T_Surge_detection:=maskbitFunction(Trip_BITs_64_to_79,0);
T_VGD_fault :=maskbitFunction(Trip_BITs_64_to_79,1);
T_Long_time_PRV :=maskbitFunction(Trip_BITs_64_to_79,2);
T_Comp_thrust_bearing_position :=maskbitFunction(Trip_BITs_64_to_79,3);
T_Comp_thrust_neg_move:=maskbitFunction(Trip_BITs_64_to_79,4);
T_Comp_thrust_pos_move:=maskbitFunction(Trip_BITs_64_to_79,5);
S_Spare_1:=maskbitFunction(Trip_BITs_64_to_79,6);
S_Spare_1:=maskbitFunction(Trip_BITs_64_to_79,7);
S_Spare_1:=maskbitFunction(Trip_BITs_64_to_79,8);
S_Spare_1:=maskbitFunction(Trip_BITs_64_to_79,9);
S_Spare_1:=maskbitFunction(Trip_BITs_64_to_79,10);
S_Spare_1:=maskbitFunction(Trip_BITs_64_to_79,11);
S_Spare_1:=maskbitFunction(Trip_BITs_64_to_79,12);
S_Spare_1:=maskbitFunction(Trip_BITs_64_to_79,13);
S_Spare_1:=maskbitFunction(Trip_BITs_64_to_79,14);
S_Spare_1:=maskbitFunction(Trip_BITs_64_to_79,15);

T_Sensor_low_signal_AI_64 :=maskbitFunction(Trip_BITs_80_to_95,0);
T_Sensor_high_signal_AI_64 :=maskbitFunction(Trip_BITs_80_to_95,1);
T_Sensor_low_signal_AI_66 :=maskbitFunction(Trip_BITs_80_to_95,2);
T_Sensor_high_signal_AI_66 :=maskbitFunction(Trip_BITs_80_to_95,3);
//T_Sensor_low_signal_AI_116:=maskbitFunction(Trip_BITs_80_to_95,4);
//T_Sensor_high_signal_AI_116:=maskbitFunction(Trip_BITs_80_to_95,5);
//T_Sensor_low_signal_AI_118:=maskbitFunction(Trip_BITs_80_to_95,6);
//T_Sensor_high_signal_AI_118:=maskbitFunction(Trip_BITs_80_to_95,7);
T_Sensor_low_signal_AI_128 :=maskbitFunction(Trip_BITs_80_to_95,8);
T_Sensor_high_signal_AI_128 :=maskbitFunction(Trip_BITs_80_to_95,9);
T_Sensor_low_signal_AI_130 :=maskbitFunction(Trip_BITs_80_to_95,10);
T_Sensor_high_signal_AI_130 :=maskbitFunction(Trip_BITs_80_to_95,11);
T_Sensor_low_signal_AI_132 :=maskbitFunction(Trip_BITs_80_to_95,12);
T_Sensor_high_signal_AI_132 :=maskbitFunction(Trip_BITs_80_to_95,13);
T_Sensor_low_signal_AI_134 :=maskbitFunction(Trip_BITs_80_to_95,14);
T_Sensor_high_signal_AI_134 :=maskbitFunction(Trip_BITs_80_to_95,15);

T_Sensor_low_signal_AI_136 :=maskbitFunction(Trip_BITs_96_to_121,0);
T_Sensor_high_signal_AI_136 :=maskbitFunction(Trip_BITs_96_to_121,1);
T_Sensor_low_signal_AI_138 :=maskbitFunction(Trip_BITs_96_to_121,2);
T_Sensor_high_signal_AI_138 :=maskbitFunction(Trip_BITs_96_to_121,3);
T_Sensor_low_signal_AI_140 :=maskbitFunction(Trip_BITs_96_to_121,4);
T_Sensor_high_signal_AI_140 :=maskbitFunction(Trip_BITs_96_to_121,5);
T_Sensor_low_signal_AI_142 :=maskbitFunction(Trip_BITs_96_to_121,6);
T_Sensor_high_signal_AI_142 :=maskbitFunction(Trip_BITs_96_to_121,7);
T_Sensor_low_signal_AI_144 :=maskbitFunction(Trip_BITs_96_to_121,8);
T_Sensor_high_signal_AI_144 :=maskbitFunction(Trip_BITs_96_to_121,9);
T_Sensor_low_signal_AI_146 :=maskbitFunction(Trip_BITs_96_to_121,10);
T_Sensor_high_signal_AI_146 :=maskbitFunction(Trip_BITs_96_to_121,11);
T_Sensor_low_signal_AI_148 :=maskbitFunction(Trip_BITs_96_to_121,12);
T_Sensor_high_signal_AI_148 :=maskbitFunction(Trip_BITs_96_to_121,13);
T_Sensor_low_signal_AI_150 :=maskbitFunction(Trip_BITs_96_to_121,14);
T_Sensor_high_signal_AI_150 :=maskbitFunction(Trip_BITs_96_to_121,15);

T_Sensor_low_signal_AI_152 :=maskbitFunction(Trip_BITs_122_to_137,0);
T_Sensor_high_signal_AI_152 :=maskbitFunction(Trip_BITs_122_to_137,1);
T_Sensor_low_signal_AI_154 :=maskbitFunction(Trip_BITs_122_to_137,2);
T_Sensor_high_signal_AI_154 :=maskbitFunction(Trip_BITs_122_to_137,3);
T_Sensor_low_signal_AI_156 :=maskbitFunction(Trip_BITs_122_to_137,4);
T_Sensor_high_signal_AI_156 :=maskbitFunction(Trip_BITs_122_to_137,5);
T_Sensor_low_signal_AI_158 :=maskbitFunction(Trip_BITs_122_to_137,6);
T_Sensor_high_signal_AI_158 :=maskbitFunction(Trip_BITs_122_to_137,7);
T_Sensor_low_signal_AI_160 :=maskbitFunction(Trip_BITs_122_to_137,8);
T_Sensor_high_signal_AI_160 :=maskbitFunction(Trip_BITs_122_to_137,9);
T_Sensor_low_signal_AI_162 :=maskbitFunction(Trip_BITs_122_to_137,10);
T_Sensor_high_signal_AI_162 :=maskbitFunction(Trip_BITs_122_to_137,11);
T_Sensor_low_signal_AI_164 :=maskbitFunction(Trip_BITs_122_to_137,12);
T_Sensor_high_signal_AI_164 :=maskbitFunction(Trip_BITs_122_to_137,13);
T_Sensor_low_signal_AI_166 :=maskbitFunction(Trip_BITs_122_to_137,14);
T_Sensor_high_signal_AI_166 :=maskbitFunction(Trip_BITs_122_to_137,15);

T_Sensor_low_signal_AI_168 :=maskbitFunction(Trip_BITs_138_to_153,0);
T_Sensor_high_signal_AI_168 :=maskbitFunction(Trip_BITs_138_to_153,1);
T_Sensor_low_signal_AI_170 :=maskbitFunction(Trip_BITs_138_to_153,2);
T_Sensor_high_signal_AI_170:=maskbitFunction(Trip_BITs_138_to_153,3);
T_Sensor_low_signal_AI_172:=maskbitFunction(Trip_BITs_138_to_153,4);
T_Sensor_high_signal_AI_172:=maskbitFunction(Trip_BITs_138_to_153,5);
T_Sensor_low_signal_AI_174:=maskbitFunction(Trip_BITs_138_to_153,6);
T_Sensor_high_signal_AI_174:=maskbitFunction(Trip_BITs_138_to_153,7);
T_Sensor_low_signal_AI_176:=maskbitFunction(Trip_BITs_138_to_153,8);
T_Sensor_high_signal_AI_176:=maskbitFunction(Trip_BITs_138_to_153,9);
T_Sensor_low_signal_AI_178:=maskbitFunction(Trip_BITs_138_to_153,10);
T_Sensor_high_signal_AI_178:=maskbitFunction(Trip_BITs_138_to_153,11);
T_Sensor_low_signal_AI_180:=maskbitFunction(Trip_BITs_138_to_153,12);
T_Sensor_high_signal_AI_180:=maskbitFunction(Trip_BITs_138_to_153,13);
T_Sensor_low_signal_AI_182:=maskbitFunction(Trip_BITs_138_to_153,14);
T_Sensor_high_signal_AI_182:=maskbitFunction(Trip_BITs_138_to_153,15);

T_Sensor_low_signal_AI_184 :=maskbitFunction(Trip_BITs_154_to_169,0);
T_Sensor_high_signal_AI_184 :=maskbitFunction(Trip_BITs_154_to_169,1);
T_Sensor_low_signal_AI_186 :=maskbitFunction(Trip_BITs_154_to_169,2);
T_Sensor_high_signal_AI_186 :=maskbitFunction(Trip_BITs_154_to_169,3);
T_Sensor_low_signal_AI_188 :=maskbitFunction(Trip_BITs_154_to_169,4);
T_Sensor_high_signal_AI_188 :=maskbitFunction(Trip_BITs_154_to_169,5);
T_Sensor_low_signal_AI_190 :=maskbitFunction(Trip_BITs_154_to_169,6);
T_Sensor_high_signal_AI_190 :=maskbitFunction(Trip_BITs_154_to_169,7);
T_Sensor_low_signal_AI_192 :=maskbitFunction(Trip_BITs_154_to_169,8);
T_Sensor_high_signal_AI_192 :=maskbitFunction(Trip_BITs_154_to_169,9);
T_Sensor_low_signal_AI_194 :=maskbitFunction(Trip_BITs_154_to_169,10);
T_Sensor_high_signal_AI_194 :=maskbitFunction(Trip_BITs_154_to_169,11);
T_Sensor_low_signal_AI_196 :=maskbitFunction(Trip_BITs_154_to_169,12);
T_Sensor_high_signal_AI_196 :=maskbitFunction(Trip_BITs_154_to_169,13);
T_Sensor_low_signal_AI_198 :=maskbitFunction(Trip_BITs_154_to_169,14);
T_Sensor_high_signal_AI_198 :=maskbitFunction(Trip_BITs_154_to_169,15);

T_Sensor_low_signal_AI_200 :=maskbitFunction(Trip_BITs_170_to_185,0);
T_Sensor_high_signal_AI_200 :=maskbitFunction(Trip_BITs_170_to_185,1);
T_Sensor_low_signal_AI_202 :=maskbitFunction(Trip_BITs_170_to_185,2);
T_Sensor_high_signal_AI_202 :=maskbitFunction(Trip_BITs_170_to_185,3);
T_Sensor_low_signal_AI_204 :=maskbitFunction(Trip_BITs_170_to_185,4);
T_Sensor_high_signal_AI_204 :=maskbitFunction(Trip_BITs_170_to_185,5);
T_Sensor_low_signal_AI_206 :=maskbitFunction(Trip_BITs_170_to_185,6);
T_Sensor_high_signal_AI_206 :=maskbitFunction(Trip_BITs_170_to_185,7);
S_Spare_1:=maskbitFunction(Trip_BITs_170_to_185,8);
S_Spare_1 :=maskbitFunction(Trip_BITs_170_to_185,9);
S_Spare_1 :=maskbitFunction(Trip_BITs_170_to_185,10);
S_Spare_1 :=maskbitFunction(Trip_BITs_170_to_185,11);
S_Spare_1 :=maskbitFunction(Trip_BITs_170_to_185,12);
S_Spare_1 :=maskbitFunction(Trip_BITs_170_to_185,13);
S_Spare_1 :=maskbitFunction(Trip_BITs_170_to_185,14);
S_Spare_1 :=maskbitFunction(Trip_BITs_170_to_185,15);

T_Transformer_winding_temp :=maskbitFunction(Trip_BITs_186_to_201,0);
T_trafo_opening_main_breaker :=maskbitFunction(Trip_BITs_186_to_201,1);
S_Spare_1 :=maskbitFunction(Trip_BITs_186_to_201,2);
S_Spare_1 :=maskbitFunction(Trip_BITs_186_to_201,3);
S_Spare_1 :=maskbitFunction(Trip_BITs_186_to_201,4);
S_Spare_1 :=maskbitFunction(Trip_BITs_186_to_201,5);
S_Spare_1 :=maskbitFunction(Trip_BITs_186_to_201,6);
S_Spare_1 :=maskbitFunction(Trip_BITs_186_to_201,7);
S_Spare_1 :=maskbitFunction(Trip_BITs_186_to_201,8);
S_Spare_1 :=maskbitFunction(Trip_BITs_186_to_201,9);
S_Spare_1 :=maskbitFunction(Trip_BITs_186_to_201,10);
S_Spare_1 :=maskbitFunction(Trip_BITs_186_to_201,11);
S_Spare_1 :=maskbitFunction(Trip_BITs_186_to_201,12);
S_Spare_1 :=maskbitFunction(Trip_BITs_186_to_201,13);
S_Spare_1 :=maskbitFunction(Trip_BITs_186_to_201,14);
S_Spare_1 :=maskbitFunction(Trip_BITs_186_to_201,15);


// Alarm bits
A_low_disch_press:=maskbitFunction(Alarm_BITs_0_to_15,0);
A_high_disch_press:=maskbitFunction(Alarm_BITs_0_to_15,1);
A_Low_suction_pressure:=maskbitFunction(Alarm_BITs_0_to_15,2);
A_High_suction_pressure:=maskbitFunction(Alarm_BITs_0_to_15,3);
A_Low_press_ratio:=maskbitFunction(Alarm_BITs_0_to_15,4);
A_High_discharge_temp :=maskbitFunction(Alarm_BITs_0_to_15,5);
A_Low_discharge_superheat:=maskbitFunction(Alarm_BITs_0_to_15,6);
A_High_discharge_superheat:=maskbitFunction(Alarm_BITs_0_to_15,7);
S_Spare_1:=maskbitFunction(Alarm_BITs_0_to_15,8);
S_Spare_1:=maskbitFunction(Alarm_BITs_0_to_15,9);
A_Low_temp_oil_inlet_comp:=maskbitFunction(Alarm_BITs_0_to_15,10);
A_High_temp_oil_inlet_comp:=maskbitFunction(Alarm_BITs_0_to_15,11);
A_Low_oil_temp_receiver:=maskbitFunction(Alarm_BITs_0_to_15,12);
A_High_oil_temp_receiver:=maskbitFunction(Alarm_BITs_0_to_15,13);
A_Low_oil_diff_pressure:=maskbitFunction(Alarm_BITs_0_to_15,14);
A_High_oil_diff_pressure:=maskbitFunction(Alarm_BITs_0_to_15,15);

A_High_oil_filter_diff_press:=maskbitFunction(Alarm_BITs_16_to_31,0);
S_Spare_1:=maskbitFunction(Alarm_BITs_16_to_31,1);
S_Spare_1:=maskbitFunction(Alarm_BITs_16_to_31,2);
A_Low_CW_outlet_temp:=maskbitFunction(Alarm_BITs_16_to_31,3);
A_High_CW_inlet_temp:=maskbitFunction(Alarm_BITs_16_to_31,4);
A_Low_CW_dP:=maskbitFunction(Alarm_BITs_16_to_31,5);
A_High_CW_dP:=maskbitFunction(Alarm_BITs_16_to_31,6);
S_Spare_1:=maskbitFunction(Alarm_BITs_16_to_31,7);
S_Spare_1:=maskbitFunction(Alarm_BITs_16_to_31,8);
A_Low_SW_inlet_temp:=maskbitFunction(Alarm_BITs_16_to_31,9);
A_High_SW_inlet_temp:=maskbitFunction(Alarm_BITs_16_to_31,10);
A_Low_SW_dP:=maskbitFunction(Alarm_BITs_16_to_31,11);
A_High_SW_dP:=maskbitFunction(Alarm_BITs_16_to_31,12);
A_Low_liquid_level:=maskbitFunction(Alarm_BITs_16_to_31,13);
A_Seawater_pump_not_running:=maskbitFunction(Alarm_BITs_16_to_31,14);
S_Spare_1:=maskbitFunction(Alarm_BITs_16_to_31,15);

S_Spare_1:=maskbitFunction(Alarm_BITs_32_to_47,0);
A_High_motor_wind_temp_R:=maskbitFunction(Alarm_BITs_32_to_47,1);
A_High_motor_wind_temp_S:=maskbitFunction(Alarm_BITs_32_to_47,2);
A_High_motor_wind_temp_T:=maskbitFunction(Alarm_BITs_32_to_47,3);
A_High_comp_mo_DE_bear_temp:=maskbitFunction(Alarm_BITs_32_to_47,4);
A_High_comp_mo_NDE_bear_temp:=maskbitFunction(Alarm_BITs_32_to_47,5);
A_High_motor_air_temp:=maskbitFunction(Alarm_BITs_32_to_47,6); 
A_High_comp_mo_DE_bear_vib:=maskbitFunction(Alarm_BITs_32_to_47,7);
A_High_comp_mo_NDE_bear_vib:=maskbitFunction(Alarm_BITs_32_to_47,8);
S_Spare_1:=maskbitFunction(Alarm_BITs_32_to_47,9);
S_Spare_1:=maskbitFunction(Alarm_BITs_32_to_47,10);
A_VGD_fault:=maskbitFunction(Alarm_BITs_32_to_47,11);
A_High_control_panel_temp:=maskbitFunction(Alarm_BITs_32_to_47,12);
A_Suction_press_limit:=maskbitFunction(Alarm_BITs_32_to_47,13);
A_Discharge_press_limit:=maskbitFunction(Alarm_BITs_32_to_47,14);
A_Discharge_superheat_limit:=maskbitFunction(Alarm_BITs_32_to_47,15);

A_Motor_current_limit:=maskbitFunction(Alarm_BITs_48_to_63,0);
S_Spare_1:=maskbitFunction(Alarm_BITs_48_to_63,1);
S_Spare_1:=maskbitFunction(Alarm_BITs_48_to_63,2);
S_Spare_1:=maskbitFunction(Alarm_BITs_48_to_63,3);
S_Spare_1:=maskbitFunction(Alarm_BITs_48_to_63,4);
S_Spare_1:=maskbitFunction(Alarm_BITs_48_to_63,5);
S_Spare_1:=maskbitFunction(Alarm_BITs_48_to_63,6);
S_Spare_1:=maskbitFunction(Alarm_BITs_48_to_63,7);
S_Spare_1:=maskbitFunction(Alarm_BITs_48_to_63,8);
S_Spare_1:=maskbitFunction(Alarm_BITs_48_to_63,9);
S_Spare_1:=maskbitFunction(Alarm_BITs_48_to_63,10);
S_Spare_1:=maskbitFunction(Alarm_BITs_48_to_63,11);
S_Spare_1:=maskbitFunction(Alarm_BITs_48_to_63,12);
S_Spare_1:=maskbitFunction(Alarm_BITs_48_to_63,13);
S_Spare_1:=maskbitFunction(Alarm_BITs_48_to_63,14);
S_Spare_1:=maskbitFunction(Alarm_BITs_48_to_63,15);

A_Transformer_winding_temp:=maskbitFunction(Alarm_BITs_64_to_79,0);
S_Spare_1:=maskbitFunction(Alarm_BITs_64_to_79,1);
S_Spare_1:=maskbitFunction(Alarm_BITs_64_to_79,2);
S_Spare_1:=maskbitFunction(Alarm_BITs_64_to_79,3);
S_Spare_1:=maskbitFunction(Alarm_BITs_64_to_79,4);
S_Spare_1:=maskbitFunction(Alarm_BITs_64_to_79,5);
S_Spare_1:=maskbitFunction(Alarm_BITs_64_to_79,6);
S_Spare_1:=maskbitFunction(Alarm_BITs_64_to_79,7);
S_Spare_1:=maskbitFunction(Alarm_BITs_64_to_79,8);
S_Spare_1:=maskbitFunction(Alarm_BITs_64_to_79,9);
S_Spare_1:=maskbitFunction(Alarm_BITs_64_to_79,10);
S_Spare_1:=maskbitFunction(Alarm_BITs_64_to_79,11);
S_Spare_1:=maskbitFunction(Alarm_BITs_64_to_79,12);
S_Spare_1:=maskbitFunction(Alarm_BITs_64_to_79,13);
S_Spare_1:=maskbitFunction(Alarm_BITs_64_to_79,14);
S_Spare_1:=maskbitFunction(Alarm_BITs_64_to_79,15);

// Statusbits
DI_0_0_Emergency_stop:=maskbitFunction(Status_BITs_0_to_15,0);
Unit_start_switch:=maskbitFunction(Status_BITs_0_to_15,1);
DI_0_2_Fault_reset:=maskbitFunction(Status_BITs_0_to_15,2);
Unit_auto:=maskbitFunction(Status_BITs_0_to_15,3);
Unit_remote:=maskbitFunction(Status_BITs_0_to_15,4);
Unit_manual:=maskbitFunction(Status_BITs_0_to_15,5);
DI_0_6_Overload_protection:=maskbitFunction(Status_BITs_0_to_15,6);
Unit_running:=maskbitFunction(Status_BITs_0_to_15,7);
DI_1_0_Overload_oilpump:=maskbitFunction(Status_BITs_0_to_15,8);
Comp_oil_pump:=maskbitFunction(Status_BITs_0_to_15,9);
Sea_water_pump:=maskbitFunction(Status_BITs_0_to_15,10);
CW_pump_running:=maskbitFunction(Status_BITs_0_to_15,11);
DI_1_4_Power_available:=maskbitFunction(Status_BITs_0_to_15,12);
DI_1_5_Starter_failure:=maskbitFunction(Status_BITs_0_to_15,13);
//CW_Pump_Remote_Start_Available:=maskbitFunction(Status_BITs_0_to_15,14);
//T_CW_Pump:=maskbitFunction(Status_BITs_0_to_15,15);

DI_8_0_Controlpanel_temp:=maskbitFunction(Status_BITs_16_to_31,0);
CW_Flow_ind:=maskbitFunction(Status_BITs_16_to_31,1);
DI_8_2_VGD_limit_switch:=maskbitFunction(Status_BITs_16_to_31,2);
DI_8_3_water_leak_motor:=maskbitFunction(Status_BITs_16_to_31,3);
DI_8_4_Catodic_protection:=maskbitFunction(Status_BITs_16_to_31,4);
DI_8_5_Trust_bearing_probe:=maskbitFunction(Status_BITs_16_to_31,5);
DI_8_6_ESD_operation:=maskbitFunction(Status_BITs_16_to_31,6);
DI_8_7:=maskbitFunction(Status_BITs_16_to_31,7);
DI_9_0_MV_breaker_available:=maskbitFunction(Status_BITs_16_to_31,8);
DI_9_1:=maskbitFunction(Status_BITs_16_to_31,9);
DI_9_2_Safe_return_to_port:=maskbitFunction(Status_BITs_16_to_31,10);
VFD_ready:=maskbitFunction(Status_BITs_16_to_31,11);
DI_9_4_VFD_emergency_stop:=maskbitFunction(Status_BITs_16_to_31,12);
Remote_bilge_pump_control:=maskbitFunction(Status_BITs_16_to_31,13);
//T_Transformer:=maskbitFunction(Status_BITs_16_to_31,14);
//A_Transformer:=maskbitFunction(Status_BITs_16_to_31,15);

DO_0_0_Start_signal_comp:=maskbitFunction(Status_BITs_32_to_47,0);
DO_0_1_Start_signal_oil_pump:=maskbitFunction(Status_BITs_32_to_47,1);
DO_0_2_Start_signal_SW_pump:=maskbitFunction(Status_BITs_32_to_47,2);
DO_0_3_Start_signal_CW_pump:=maskbitFunction(Status_BITs_32_to_47,3);
DO_0_4_Solenoid_valve_oil:=maskbitFunction(Status_BITs_32_to_47,4);
DO_0_5_Solenoid_valve_liquid:=maskbitFunction(Status_BITs_32_to_47,5);
DO_0_6_Oil_heater:=maskbitFunction(Status_BITs_32_to_47,6);
DO_0_7_Comp_heater:=maskbitFunction(Status_BITs_32_to_47,7);
DO_1_0:=maskbitFunction(Status_BITs_32_to_47,8);
DO_1_1:=maskbitFunction(Status_BITs_32_to_47,9);
S_Spare_1:=maskbitFunction(Status_BITs_32_to_47,10);
S_Spare_1:=maskbitFunction(Status_BITs_32_to_47,11);
S_Spare_1:=maskbitFunction(Status_BITs_32_to_47,12);
S_Spare_1:=maskbitFunction(Status_BITs_32_to_47,13);
S_Spare_1:=maskbitFunction(Status_BITs_32_to_47,14);
S_Spare_1:=maskbitFunction(Status_BITs_32_to_47,15);

DO_8_0_Liquid_valve_open:=maskbitFunction(Status_BITs_48_to_63,0);
DO_8_1_Liquid_valve_close:=maskbitFunction(Status_BITs_48_to_63,1);
DO_8_2_VGD_open:=maskbitFunction(Status_BITs_48_to_63,2);
DO_8_3_VGD_close:=maskbitFunction(Status_BITs_48_to_63,3);
DO_8_4_PRV_open:=maskbitFunction(Status_BITs_48_to_63,4);
DO_8_5_PRV_close:=maskbitFunction(Status_BITs_48_to_63,5);
DO_8_6_HGV_open:=maskbitFunction(Status_BITs_48_to_63,6);
DO_8_7_HGV_close:=maskbitFunction(Status_BITs_48_to_63,7);
DO_9_0_Main_breaker_ready:=maskbitFunction(Status_BITs_48_to_63,8);
DO_9_1_Close_order_swv_overboard:=maskbitFunction(Status_BITs_48_to_63,9);
DO_9_2_Open_order_swv_bypass:=maskbitFunction(Status_BITs_48_to_63,10);
DO_9_3_Close_order_swv_bypass:=maskbitFunction(Status_BITs_48_to_63,11);
DO_9_4:=maskbitFunction(Status_BITs_48_to_63,12);
DO_9_5:=maskbitFunction(Status_BITs_48_to_63,13);
DO_9_6:=maskbitFunction(Status_BITs_48_to_63,14);
DO_9_7:=maskbitFunction(Status_BITs_48_to_63,15);

DO_12_0_Power_request:=maskbitFunction(Status_BITs_64_to_79,0);
DO_12_1_Compressor_ready:=maskbitFunction(Status_BITs_64_to_79,1);
Unit_trip:=maskbitFunction(Status_BITs_64_to_79,2);
Unit_alarm:=maskbitFunction(Status_BITs_64_to_79,3);
DO_12_4_Control_panel_alarm:=maskbitFunction(Status_BITs_64_to_79,4);
DO_12_5_Auto_reset:=maskbitFunction(Status_BITs_64_to_79,5);
DO_12_6_Unit_running:=maskbitFunction(Status_BITs_64_to_79,6);
//DO_12_7_Emergency_MV_Breaker:=maskbitFunction(Status_BITs_64_to_79,7);
T_Spare_3:=maskbitFunction(Status_BITs_64_to_79,8);
T_Spare_3:=maskbitFunction(Status_BITs_64_to_79,9);
T_Spare_3:=maskbitFunction(Status_BITs_64_to_79,10);
T_Spare_3:=maskbitFunction(Status_BITs_64_to_79,11);
T_Spare_3:=maskbitFunction(Status_BITs_64_to_79,12);
T_Spare_3:=maskbitFunction(Status_BITs_64_to_79,13);
T_Spare_3:=maskbitFunction(Status_BITs_64_to_79,14);
T_Spare_3:=maskbitFunction(Status_BITs_64_to_79,15);

Unit_manual:=maskbitFunction(Status_BITs_80_to_95,0);
Unit_available:=maskbitFunction(Status_BITs_80_to_95,1);
CW_Flow_ind:=maskbitFunction(Status_BITs_80_to_95,2);
Start_inhib_time_Oil_receiver_temp:=maskbitFunction(Status_BITs_80_to_95,3);
Start_inhib_time_between_Stop_Start:=maskbitFunction(Status_BITs_80_to_95,4);
Start_inhib_time_between_Start:=maskbitFunction(Status_BITs_80_to_95,5);
Start_inhib_PRV_not_min:=maskbitFunction(Status_BITs_80_to_95,6);
VFD_ramp_100_perc:=maskbitFunction(Status_BITs_80_to_95,7);
VFD_locked_100_perc:=maskbitFunction(Status_BITs_80_to_95,8);
VFD_ramp_d_PRVcontrol:=maskbitFunction(Status_BITs_80_to_95,9);
PRV_control:=maskbitFunction(Status_BITs_80_to_95,10);
VFD_control:=maskbitFunction(Status_BITs_80_to_95,11);
VFD_fixed_speed:=maskbitFunction(Status_BITs_80_to_95,12);
T_Spare_3:=maskbitFunction(Status_BITs_80_to_95,13);
T_Spare_3:=maskbitFunction(Status_BITs_80_to_95,14);
T_Spare_3:=maskbitFunction(Status_BITs_80_to_95,15);


// Graphic controls
IF Unit_remote THEN
	Unit_switch_status:=2;
ELSIF Unit_auto THEN 
	Unit_switch_status:=3;
ELSIF Unit_manual THEN 
	Unit_switch_status:=4;

END_IF ;	

IF select_trendvalue > 0 THEN
	show_trendvalue[select_trendvalue]:= TRUE;
ELSIF select_trendvalue = 0 THEN
	FOR i := 0 TO 50 DO
      show_trendvalue[i] := FALSE;
   	END_FOR
END_IF ;

END_PROGRAM

// Calculus
PROGRAM Calculus
VAR


// MWCC

NakW_chiller_3 : REAL ;
NakW_chiller_4 : REAL ;

COP_chiller_3 : REAL ;
COP_chiller_4 : REAL ;
NakW_chiller_5 : REAL ;
NakW_chiller_6 : REAL ;

COP_chiller_5 : REAL ;
COP_chiller_6 : REAL ;
{attribute 'ac_datalog_hysteresis' := '100'}
{attribute 'ac_datalog' := 'DatalogChannel'}
Tot_Power_motor : REAL ;
{attribute 'ac_datalog_hysteresis' := '300'}
{attribute 'ac_datalog' := 'DatalogChannel'}
Tot_Q2 : REAL ;
{attribute 'ac_datalog_hysteresis' := '100'}
{attribute 'ac_datalog' := 'DatalogChannel'}
Tot_Q2_MWh : REAL ;
{attribute 'ac_datalog_hysteresis' := '100'}
{attribute 'ac_datalog' := 'DatalogChannel'}
Tot_P1_MWh : REAL ;
Power_motor_3_kW : REAL ;
Power_motor_4_kW : REAL ;
Power_motor_5_kW : REAL ;
Power_motor_6_kW : REAL ;
Power_3_not_zero : REAL ;
Power_4_not_zero : REAL ;
Power_5_not_zero : REAL ;
Power_6_not_zero : REAL ;

// SE700
Q2kW_chiller_1 : REAL ;
Q2kW_chiller_2 : REAL ;
Chiller_1_dpCW_bar : REAL ;
Chiller_2_dpCW_bar : REAL ;
Chiller_1_SR_dpCW_bar : REAL ;
Chiller_2_SR_dpCW_bar : REAL ;
Power_motor_1_kW : REAL ;
Power_motor_2_kW : REAL ;
Power_1_not_zero : REAL ;
Power_2_not_zero : REAL ;
NakW_chiller_1 : REAL ;
NakW_chiller_2 : REAL ;
COP_chiller_1 : REAL ;
COP_chiller_2 : REAL ;



Power_3_not_zero_func: WORD := 100;
Power_4_not_zero_func :  WORD := 100;
COP_chiller_3_func :  WORD := 100;
COP_chiller_4_func :  WORD := 100;
Power_5_not_zero_func: WORD := 100;
Power_6_not_zero_func :  WORD := 100;
COP_chiller_5_func :  WORD := 100;
COP_chiller_6_func :  WORD := 100;
Tot_Power_motor_func :  WORD := 100;
Tot_Q2_func :  WORD := 100;
Tot_Q2_MWh_func :  WORD := 100;
Tot_Na_MWh_func :  WORD := 100;
Power_motor_3_kW_func :  WORD := 100;
Power_motor_4_kW_func :  WORD := 100;

// SE700

Man_Auto_Chiller_1_func :  WORD := 100;
Man_Auto_Chiller_2_func :  WORD := 100;
//SE700_Chiller_1_Modb|||VALISERR(LOCAL.MODBUS2.Chiller_1.Program_number);//
//SE700_Chiller_2_Modb|||VALISERR(LOCAL.MODBUS2.Chiller_2.Program_number);
Flow_factor_chiller1_func :  WORD := 100;
Flow_factor_chiller2_func :  WORD := 100;


SR_Nom_dP_bar_func :  WORD := 100;


Chiller_1_dT_func :  WORD := 100;
Chiller_2_dT_func :  WORD := 100;
Chiller_1_max_dT_func :  WORD := 100;
Chiller_2_max_dT_func :  WORD := 100;
Chiller_1_Capacity_func :  WORD := 100;
Chiller_2_Capacity_func :  WORD := 100;
Chiller_1_CapacitykW_func :  WORD := 100;
Chiller_2_CapacitykW_func :  WORD := 100;
Chiller_1_dpCW_bar_func :  WORD := 100;
Chiller_2_dpCW_bar_func :  WORD := 100;
Chiller_1_SR_dpCW_bar_func :  WORD := 100;
Chiller_2_SR_dpCW_bar_func :  WORD := 100;
Power_motor_1_kW_func :  WORD := 100;
Power_motor_2_kW_func :  WORD := 100;
Power_1_not_zero_func :  WORD := 100;
Power_2_not_zero_func :  WORD := 100;
COP_chiller_1_func :  WORD := 100;
COP_chiller_2_func :  WORD := 100;
Chiller_1_Capacity_corr_flow_factor_func :  WORD := 100;
Chiller_2_Capacity_corr_flow_factor_func :  WORD := 100;
// New Variables
PI_chiller_1  : REAL ;
PI_chiller_1_word : WORD ;
PI_Calc_Error_AC1 : BOOL ;
PI_chiller_2  : REAL ;
PI_chiller_2_word : WORD ;
PI_Calc_Error_AC2 : BOOL ;
PI_chiller_3  : REAL ;
PI_chiller_3_word : WORD ;
PI_Calc_Error_AC3 : BOOL ;
PI_chiller_4  : REAL ;
PI_chiller_4_word : WORD ;
PI_Calc_Error_AC4 : BOOL ;
PI_chiller_5  : REAL ;
PI_chiller_5_word : WORD ;
PI_Calc_Error_AC5 : BOOL ;
PI_chiller_6  : REAL ;
PI_chiller_6_word : WORD ;
PI_Calc_Error_AC6 : BOOL ;
delaytimer2 : TON ;	
resetbuttons : BOOL := FALSE  ;
COP_theo_AC1 :REAL ;	
COP_theo_AC2 :REAL ;
COP_theo_AC3 :REAL ;
COP_theo_AC4 :REAL ;
COP_theo_AC5 :REAL ;
COP_theo_AC6 :REAL ;
totRunningChillers : INT;
WastedEnergy_AC1 :REAL ;
WastedEnergy_AC1_word :WORD ;
WastedEnergy_AC2 :REAL ;
WastedEnergy_AC2_word :WORD ;
WastedEnergy_AC3 :REAL ;
WastedEnergy_AC3_word :WORD ;
WastedEnergy_AC4 :REAL ;
WastedEnergy_AC4_word :WORD ;
WastedEnergy_AC5 :REAL ;
WastedEnergy_AC5_word :WORD ;
WastedEnergy_AC6 :REAL ;
WastedEnergy_AC6_word :WORD ;
Total_PI : REAL ;
// Time variables
Result_time : SysTimeRtc.RTS_IEC_RESULT;
udiLocal_DateAndTime : UDINT;
current_date : UDINT ;

	
END_VAR

IF GVL.startUp THEN
	startupReadcsv();
	IF NOT GVL.startUp THEN	
		GVL.xReadCOP := FALSE;
		GVL.startdelaytimer :=TRUE;
	END_IF
	
END_IF

GVL.delaytimer (IN:= GVL.startdelaytimer, PT:=T#5S);
IF GVL.delaytimer.Q THEN
	GVL.xReadCOP := TRUE;
	GVL.startdelaytimer:=FALSE;
	resetbuttons := TRUE ;
END_IF
delaytimer2 (IN:= resetbuttons, PT:=T#5S);
IF delaytimer2.Q THEN
	GVL.xReadCOP := FALSE;
	GVL.initRead := FALSE;
	resetbuttons := FALSE;
END_IF

// Get system time
current_date := TO_UDINT(SysTimeRtcGet(Result_time));
Result_time := SysTimeRTCConvertUTCToLocal(current_date, udiLocal_DateAndTime);
GVL.CurrentDate := TO_DT(udiLocal_DateAndTime); // DT#2018-6-6-9:8:38

// MWCC
Tot_Q2_MWh:=Tot_Q2:=Chiller_1.Q2_chillerMWh + Chiller_2.Q2_chillerMWh + Chiller_3.Q2_chillerMWh + Chiller_4.Q2_chillerMWh + Chiller_5.Q2_chillerMWh (* + Chiller_6.Q2_chillerMWh*) ;
//Tot_Q2_MWh:=Tot_Q2:=Sequence.Chiller_1_Q2_MWh + Sequence.Chiller_2_Q2_MWh + Sequence.Chiller_3_Q2_MWh + Sequence.Chiller_4_Q2_MWh + Sequence.Chiller_5_Q2_MWh + Sequence.Chiller_6_Q2_MWh ;
Tot_P1_MWh:=Tot_Q2:=Chiller_1.Chiller_P1_MWh + Chiller_2.Chiller_P1_MWh + Chiller_3.Chiller_P1_MWh + Chiller_4.Chiller_P1_MWh + Chiller_5.Chiller_P1_MWh (* + Chiller_6.Chiller_P1_MWh*) ;
//Tot_P1_MWh:=Tot_Q2:=Sequence.Chiller_1_P1_MWh + Sequence.Chiller_2_P1_MWh + Sequence.Chiller_3_P1_MWh + Sequence.Chiller_4_P1_MWh + Sequence.Chiller_5_P1_MWh + Sequence.Chiller_6_P1_MWh ;

// New Func
Power_motor_1_kW:=Chiller_1.P1_motor_kW;
Power_motor_2_kW:=Chiller_2.P1_motor_kW;
Power_motor_3_kW:=Chiller_3.P1_motor_kW;
Power_motor_4_kW:=Chiller_4.P1_motor_kW;
Power_motor_5_kW:=Chiller_5.P1_motor_kW;
//Power_motor_6_kW:=Chiller_6.P1_motor_kW;

Tot_Power_motor:=Power_motor_1_kW + Power_motor_2_kW + Power_motor_3_kW + Power_motor_4_kW + Power_motor_5_kW (* + Power_motor_6_kW*);
//Tot_Q2:=sequence.Q2kW_chiller_1 + sequence.Q2kW_chiller_2 + Sequence.Q2kW_chiller_3 + Sequence.Q2kW_chiller_4 + Sequence.Q2kW_chiller_5 + Sequence.Q2kW_chiller_6;
Tot_Q2:=Chiller_1.Chiller_capacity_kW + Chiller_2.Chiller_capacity_kW + Chiller_3.Chiller_capacity_kW + Chiller_4.Chiller_capacity_kW + Chiller_5.Chiller_capacity_kW (* + Chiller_6.Chiller_capacity_kW*);
COP_chiller_1:=Chiller_1.COP_chiller_ele;
COP_chiller_2:=Chiller_2.COP_chiller_ele;
COP_chiller_3:=Chiller_3.COP_chiller_ele;
COP_chiller_4:=Chiller_4.COP_chiller_ele;
COP_chiller_5:=Chiller_5.COP_chiller_ele;
(*COP_chiller_6:=Chiller_6.COP_chiller_ele;*)

totRunningChillers := BOOL_TO_INT(Chiller_1.Unit_running) + BOOL_TO_INT(Chiller_2.Unit_running) + BOOL_TO_INT(Chiller_3.Unit_running) + BOOL_TO_INT(Chiller_4.Unit_running) + BOOL_TO_INT(Chiller_5.Unit_running) (*+ BOOL_TO_INT(Chiller_6.Unit_running)*);

IF Chiller_1.Unit_running THEN
	PI_calculation(Chiller_1.Chiller_capacity,Chiller_1.Temp_water_inlet_cond,COP_chiller_1,Chiller_1.Temp_chilled_medium_out, 1, PI_act=>PI_chiller_1, noCalc_error=>PI_Calc_Error_AC1, COP_theo=>COP_theo_AC1);	
	WastedEnergy_AC1 := Wasted_calc(Chiller_1.Chiller_capacity_kW, COP_theo_AC1, Power_motor_1_kW) ;
	ELSE
	PI_chiller_1 := 0;
	WastedEnergy_AC1 := 0;
	PI_Calc_Error_AC1 := TRUE;
	COP_theo_AC1 := 0;
END_IF

IF Chiller_2.Unit_running THEN
	PI_calculation(Chiller_2.Chiller_capacity,Chiller_2.Temp_water_inlet_cond,COP_chiller_2,Chiller_2.Temp_chilled_medium_out, 1, PI_act=>PI_chiller_2,noCalc_error=>PI_Calc_Error_AC2, COP_theo=>COP_theo_AC2);
	WastedEnergy_AC2 := Wasted_calc(Chiller_2.Chiller_capacity_kW, COP_theo_AC2, Power_motor_2_kW) ;
	ELSE
	PI_chiller_2 := 0;
	WastedEnergy_AC2 := 0;
	PI_Calc_Error_AC2 := TRUE;
	COP_theo_AC2 := 0;
END_IF

IF Chiller_3.Unit_running THEN
	PI_calculation(Chiller_3.Chiller_capacity,Chiller_3.Temp_water_inlet_cond,COP_chiller_3,Chiller_3.Temp_chilled_medium_out, 2, PI_act=>PI_chiller_3,noCalc_error=>PI_Calc_Error_AC3, COP_theo=>COP_theo_AC3);
	WastedEnergy_AC3 := Wasted_calc(Chiller_3.Chiller_capacity_kW, COP_theo_AC3, Power_motor_3_kW) ;
	ELSE
	PI_chiller_3 := 0;
	WastedEnergy_AC3 := 0;	
	PI_Calc_Error_AC3 := TRUE;
	COP_theo_AC3 := 0;
END_IF

IF Chiller_4.Unit_running THEN
	PI_calculation(Chiller_4.Chiller_capacity,Chiller_4.Temp_water_inlet_cond,COP_chiller_4,Chiller_4.Temp_chilled_medium_out, 1, PI_act=>PI_chiller_4,noCalc_error=>PI_Calc_Error_AC4, COP_theo=>COP_theo_AC4);
	WastedEnergy_AC4 := Wasted_calc(Chiller_4.Chiller_capacity_kW, COP_theo_AC4, Power_motor_4_kW) ;
	ELSE
	PI_chiller_4 := 0;
	WastedEnergy_AC4 := 0;
	PI_Calc_Error_AC4 := TRUE;
	COP_theo_AC4 := 0;
END_IF


IF Chiller_5.Unit_running THEN
	PI_calculation(Chiller_5.Chiller_capacity,Chiller_5.Temp_water_inlet_cond,COP_chiller_5,Chiller_5.Temp_chilled_medium_out, 1, PI_act=>PI_chiller_5,noCalc_error=>PI_Calc_Error_AC5, COP_theo=>COP_theo_AC5);
	WastedEnergy_AC5 := Wasted_calc(Chiller_5.Chiller_capacity_kW, COP_theo_AC5, Power_motor_5_kW) ;
	ELSE
	PI_chiller_5 := 0;
	WastedEnergy_AC5 := 0;
	PI_Calc_Error_AC5 := TRUE ;
	COP_theo_AC5 := 0;			
END_IF


(*
IF Chiller_6.Unit_running THEN
	PI_calculation(Chiller_6.Chiller_capacity,Chiller_6.Temp_water_inlet_cond,COP_chiller_6,Chiller_6.Temp_chilled_medium_out, 2, PI_act=>PI_chiller_6,noCalc_error=>PI_Calc_Error_AC6, COP_theo=>COP_theo_AC6);
	WastedEnergy_AC6 := Wasted_calc(sequence.Q2kW_chiller_6, COP_theo_AC6, Power_motor_6_kW) ;
	ELSE
	PI_chiller_6 := 0;
	WastedEnergy_AC6 := 0 ;
	PI_Calc_Error_AC6 := TRUE ;
	COP_theo_AC6 := 0;			
END_IF
*)


PI_chiller_1_word := REAL_TO_WORD(PI_chiller_1 * 100) ;
PI_chiller_2_word := REAL_TO_WORD(PI_chiller_2 * 100) ;
PI_chiller_3_word := REAL_TO_WORD(PI_chiller_3 * 100) ;
PI_chiller_4_word := REAL_TO_WORD(PI_chiller_4 * 100) ;
PI_chiller_5_word := REAL_TO_WORD(PI_chiller_5 * 100) ;
PI_chiller_6_word := REAL_TO_WORD(PI_chiller_6 * 100) ;

WastedEnergy_AC1_word := REAL_TO_WORD(WastedEnergy_AC1) ;
WastedEnergy_AC2_word := REAL_TO_WORD(WastedEnergy_AC2) ;
WastedEnergy_AC3_word := REAL_TO_WORD(WastedEnergy_AC3) ;
WastedEnergy_AC4_word := REAL_TO_WORD(WastedEnergy_AC4) ;
WastedEnergy_AC5_word := REAL_TO_WORD(WastedEnergy_AC5) ;
WastedEnergy_AC6_word := REAL_TO_WORD(WastedEnergy_AC6) ;



(*
PI_calculation(95,31,4.5,6.1, 1, PI_act=>PI_chiller_1 ,noCalc_error=>PI_Calc_Error_AC1, COP_theo=>COP_theo_AC1);
PI_calculation(92,31,4.5,6.1, 3, PI_act=>PI_chiller_2 ,noCalc_error=>PI_Calc_Error_AC2, COP_theo=>COP_theo_AC2);
PI_calculation(91,31,4.5,6.1, 2, PI_act=>PI_chiller_3 ,noCalc_error=>PI_Calc_Error_AC3, COP_theo=>COP_theo_AC3);
PI_calculation(90,31,4.5,6.1, 3, PI_act=>PI_chiller_4 ,noCalc_error=>PI_Calc_Error_AC4, COP_theo=>COP_theo_AC4);
*)

IF totRunningChillers>0 THEN
	Total_PI:=Tot_PI(PI_chiller_1, PI_chiller_2, PI_chiller_3, PI_chiller_4, PI_chiller_5, PI_chiller_6 , totRunningChillers) ;
	ELSE 
	Total_PI := 0 ;
END_IF

END_PROGRAM

// csvRead
// CSV Reader examples
PROGRAM csvRead
VAR

	
	// 'ReadAll' example
	csvReaderInit3			: CSV.CSVReaderInit;
	csvReaderInit3COP		: CSV.CSVReaderInit;
	csvReaderInit3_1		: CSV.CSVReaderInit;
	csvReaderInit3_2		: CSV.CSVReaderInit;
	csvReaderInit3_3		: CSV.CSVReaderInit;
	xRead				: BOOL;
	xRead1				: BOOL;
	xRead2				: BOOL;
	xRead3				: BOOL;
	xReadCOP			: BOOL;
	readAll				: CSV.ReadAll;
	readAllCOP	    	: CSV.ReadAll;
	//COP Adj Array	
	// {attribute 'ac_persist' := 'PersistenceChannel'}
	// saDataArray			: ARRAY[0..8, 0..80] OF STRING(100);
	asDataArray			: ARRAY[0..730] OF STRING(100);
	pasDataArray		: POINTER TO ARRAY[0..730] OF STRING(100) := ADR(asDataArray);
	asDataArray1		: ARRAY[0..730] OF STRING(100);
	pasDataArray1		: POINTER TO ARRAY[0..730] OF STRING(100) := ADR(asDataArray1);
	asDataArray2		: ARRAY[0..730] OF STRING(100);
	pasDataArray2		: POINTER TO ARRAY[0..730] OF STRING(100) := ADR(asDataArray2);
	asDataArray3		: ARRAY[0..730] OF STRING(100);
	pasDataArray3		: POINTER TO ARRAY[0..730] OF STRING(100) := ADR(asDataArray3);
	//COP Adj Array
	// {attribute 'ac_persist' := 'PersistenceChannel'}
	// saCOPDataArray			: ARRAY[0..2, 0..320] OF STRING(100);
	asCOPDataArray		: ARRAY[0..970] OF STRING(100);
	pasCOPDataArray		: POINTER TO ARRAY[0..970] OF STRING(100) := ADR(asCOPDataArray);
	//  General variables
	dataConvert			: ConvertDataArray;
	dataConvert1		: ConvertDataArray_1;
	dataConvert2		: ConvertDataArray_2;
	dataConvert3		: ConvertDataArray_3;
	dataConvert4		: ConvertDataArray_4;
	R_TRIG_0			: R_TRIG;
	R_TRIG_1			: R_TRIG;
	R_TRIG_2			: R_TRIG;
	R_TRIG_3			: R_TRIG;
	R_TRIG_4			: R_TRIG;
	{attribute 'ac_persist' := 'PersistenceChannel'}
	PIfilename1			: STRING := '/home/jci/PIcsvfiles/Britannia_4600.csv' ;
	{attribute 'ac_persist' := 'PersistenceChannel'}
	PIfilename2			: STRING := '/home/jci/PIcsvfiles/Britannia_2300.csv' ;
	{attribute 'ac_persist' := 'PersistenceChannel'}
	PIfilename3			: STRING := '/home/jci/PIcsvfiles/' ;
	{attribute 'ac_persist' := 'PersistenceChannel'}
	PIfilename4			: STRING := '/home/jci/PIcsvfiles/' ;
	{attribute 'ac_persist' := 'PersistenceChannel'}
	copAdjfilename		: STRING := '/home/jci/PIcsvfiles/COP_adj.csv' ;
	initRead			: BOOL:= FALSE ;
	convFinished		: BOOL:= FALSE ;
	
END_VAR

// Read COP adj csv file
csvReaderInit3COP(xExecute := GVL.initRead, szFileName := copAdjfilename, sLineSeparator := '$L'); // CSV.CSVReaderInit
// Convert the data array for the visualization
// Convert the data array for the visualization
readAllCOP(
    xExecute := csvReaderInit3COP.xDone AND GVL.xReadCOP,
    udiMaxElementLength := 100,
    csvReaderInit := csvReaderInit3COP,
    pasDataArray := pasCOPDataArray); // CSV.ReadAll
R_TRIG_1(CLK := readAllCOP.xDone); // R_TRIG
dataConvert1(xExecute := R_TRIG_1.Q, asData := asCOPDataArray); // ConvertDataArray_1
// Read PI file
csvReaderInit3(xExecute := GVL.initRead, szFileName := PIfilename1, sLineSeparator := '$L'); // CSV.CSVReaderInit
readAll(
    xExecute := csvReaderInit3.xDone AND GVL.xRead,
    udiMaxElementLength := 100,
    csvReaderInit := csvReaderInit3,
    pasDataArray := pasDataArray); // CSV.ReadAll
GVL.saCOPDataArray := dataConvert1.asConvertedCOPData;
R_TRIG_0(CLK := readAll.xDone); // R_TRIG
dataConvert(xExecute := R_TRIG_0.Q, asData := asDataArray); // ConvertDataArray
// Read PI file4
csvReaderInit3_3(xExecute := GVL.initRead, szFileName := PIfilename4, sLineSeparator := '$L'); // CSV.CSVReaderInit
// Convert the data array for the visualization
// Convert the data array for the visualization
readAll(
    xExecute := csvReaderInit3_3.xDone AND GVL.xRead3,
    udiMaxElementLength := 100,
    csvReaderInit := csvReaderInit3_3,
    pasDataArray := pasDataArray3); // CSV.ReadAll
R_TRIG_4(CLK := readAll.xDone); // R_TRIG
dataConvert4(xExecute := R_TRIG_4.Q, asData := asDataArray3); // ConvertDataArray_4
GVL.saDataArray3 := dataConvert4.asConvertedData;
// Convert the data array for the visualization
convFinished := dataConvert1.convert_finished;
// Read PI file3
csvReaderInit3_2(xExecute := GVL.initRead, szFileName := PIfilename3, sLineSeparator := '$L'); // CSV.CSVReaderInit
// Convert the data array for the visualization
// Convert the data array for the visualization
readAll(
    xExecute := csvReaderInit3_2.xDone AND GVL.xRead2,
    udiMaxElementLength := 100,
    csvReaderInit := csvReaderInit3_2,
    pasDataArray := pasDataArray2); // CSV.ReadAll
R_TRIG_3(CLK := readAll.xDone); // R_TRIG
dataConvert3(xExecute := R_TRIG_3.Q, asData := asDataArray2); // ConvertDataArray_3
GVL.saDataArray2 := dataConvert3.asConvertedData;
// Read PI file 2
csvReaderInit3_1(xExecute := GVL.initRead, szFileName := PIfilename2, sLineSeparator := '$L'); // CSV.CSVReaderInit
// Convert the data array for the visualization
readAll(
    xExecute := csvReaderInit3_1.xDone AND GVL.xRead1,
    udiMaxElementLength := 100,
    csvReaderInit := csvReaderInit3_1,
    pasDataArray := pasDataArray1); // CSV.ReadAll
R_TRIG_2(CLK := readAll.xDone); // R_TRIG
dataConvert2(xExecute := R_TRIG_2.Q, asData := asDataArray1); // ConvertDataArray_2
GVL.saDataArray1 := dataConvert2.asConvertedData;
GVL.saDataArray := dataConvert.asConvertedData;

END_PROGRAM

// /Alarm_list
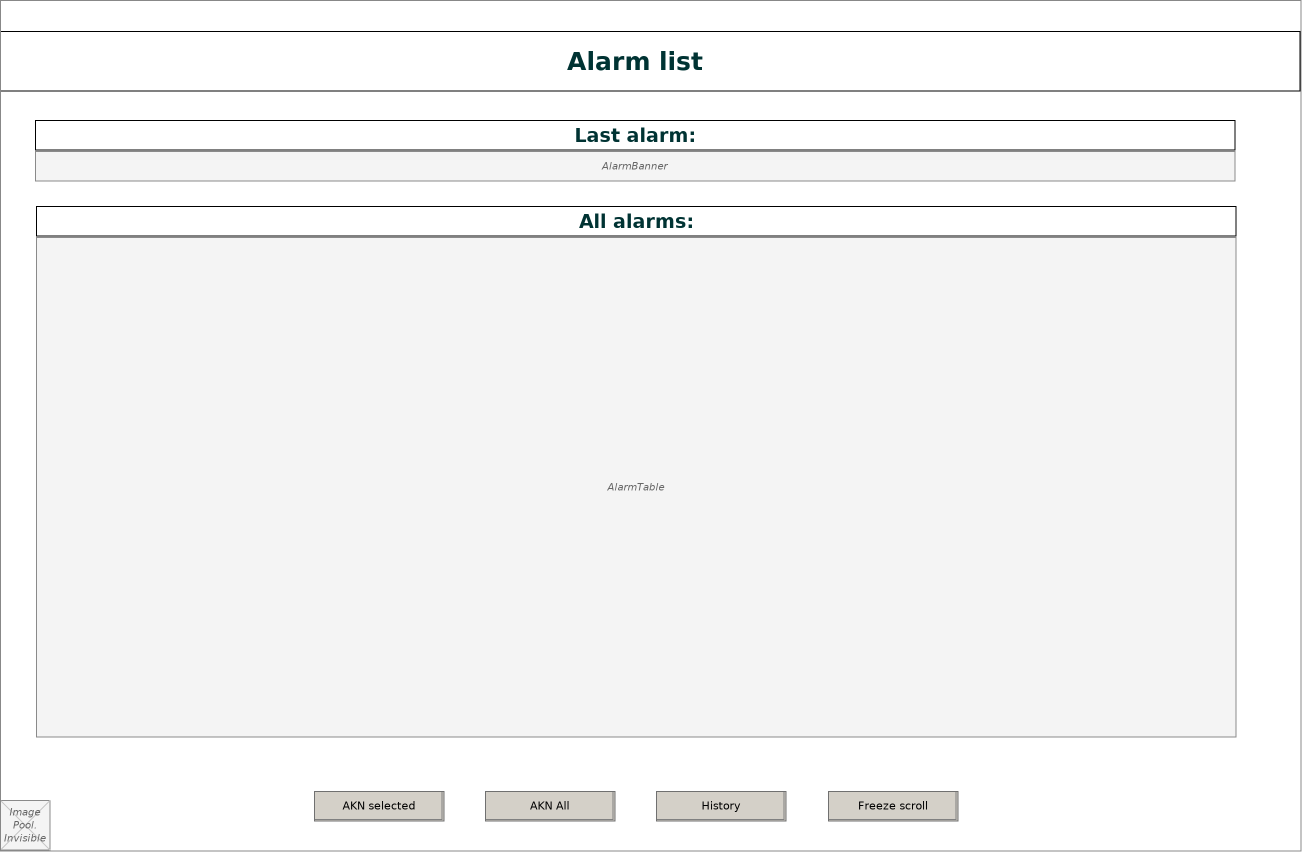
VISUALIZATION Alarm_list  // 1302x852
VAR
	AlarmACKButton : BOOL;
	AlarmACKAllButton : BOOL;
	AlarmHistoryButton : BOOL;
	AlarmFreezeButton : BOOL;
END_VAR
    AlarmTable (36,237 1200x500)
        p1521930926: __All
        p1663851261: __All
        p428520879: AlarmACKButton
        p2607059081: AlarmACKAllButton
        p3266827225: AlarmHistoryButton
        p3894972949: AlarmFreezeButton
    Button (314,791 130x30), "AKN selected"
        tap AlarmACKButton
    Button (485,791 130x30), "AKN All"
        tap AlarmACKAllButton
    Button (828,791 130x30), "Freeze scroll"
        toggle AlarmFreezeButton
    Button (656,791 130x30), "History"
        toggle AlarmHistoryButton
    Rectangle (0,31 1300x60)
    Label (247,33 776x56), "Alarm list"
    Rectangle (36,206 1200x30)
    Label (391,209 491x25), "All alarms:"
    Image (0,800 50x50), image: ImagePool.Invisible
    Rectangle (35,120 1200x30)
    Label (390,123 491x25), "Last alarm:"
    AlarmBanner (35,151 1200x30)
        p1521930926: __All
        p1663851261: __All
END_VISUALIZATION

// /Chiller1Menu
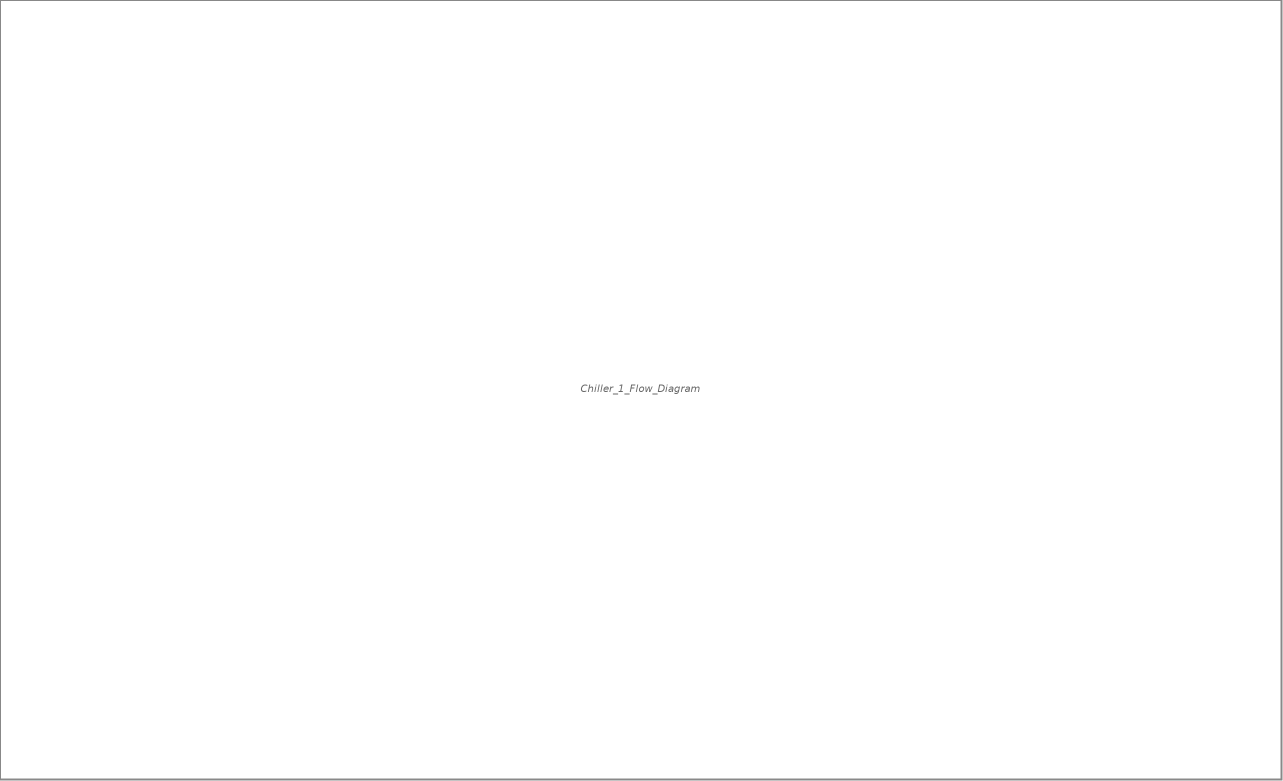
VISUALIZATION Chiller1Menu  // 1283x781
    TabControl (0,-2 1281x781)
        shows Chiller_1_Flow_Diagram()
        shows Chiller_1_Values()
        shows Chiller_1_Oil()
        shows Chiller_1_Alarm()
        shows Chiller_1_Trip()
        shows TrendMenu()
        shows Chiller_1_VFD()
        [0]: TabTitle=Diagram
        [1]: TabTitle=Measured values
        [2]: TabTitle=Oil system
        [3]: TabTitle=Alarm
        [4]: TabTitle=Trip
        [6]: TabTitle=Trend menu
END_VISUALIZATION

// /Chiller2Menu
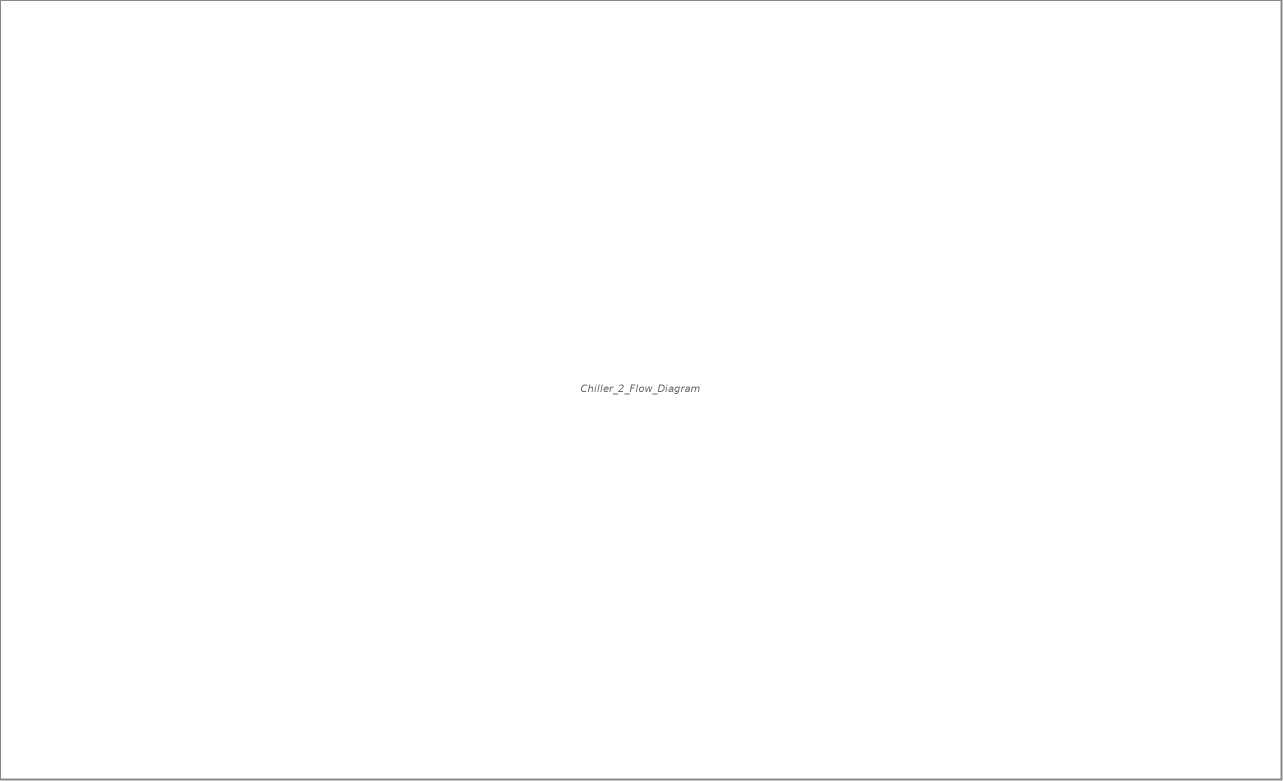
VISUALIZATION Chiller2Menu  // 1283x781
    TabControl (0,-2 1281x781)
        shows Chiller_2_Flow_Diagram()
        shows Chiller_2_Values()
        shows Chiller_2_Oil()
        shows Chiller_2_Alarm()
        shows Chiller_2_Trip()
        shows Chiller_2_VFD()
        [0]: TabTitle=Diagram
        [1]: TabTitle=Measured values
        [2]: TabTitle=Oil system
        [3]: TabTitle=Alarm
        [4]: TabTitle=Trip
END_VISUALIZATION

// /Chiller3Menu
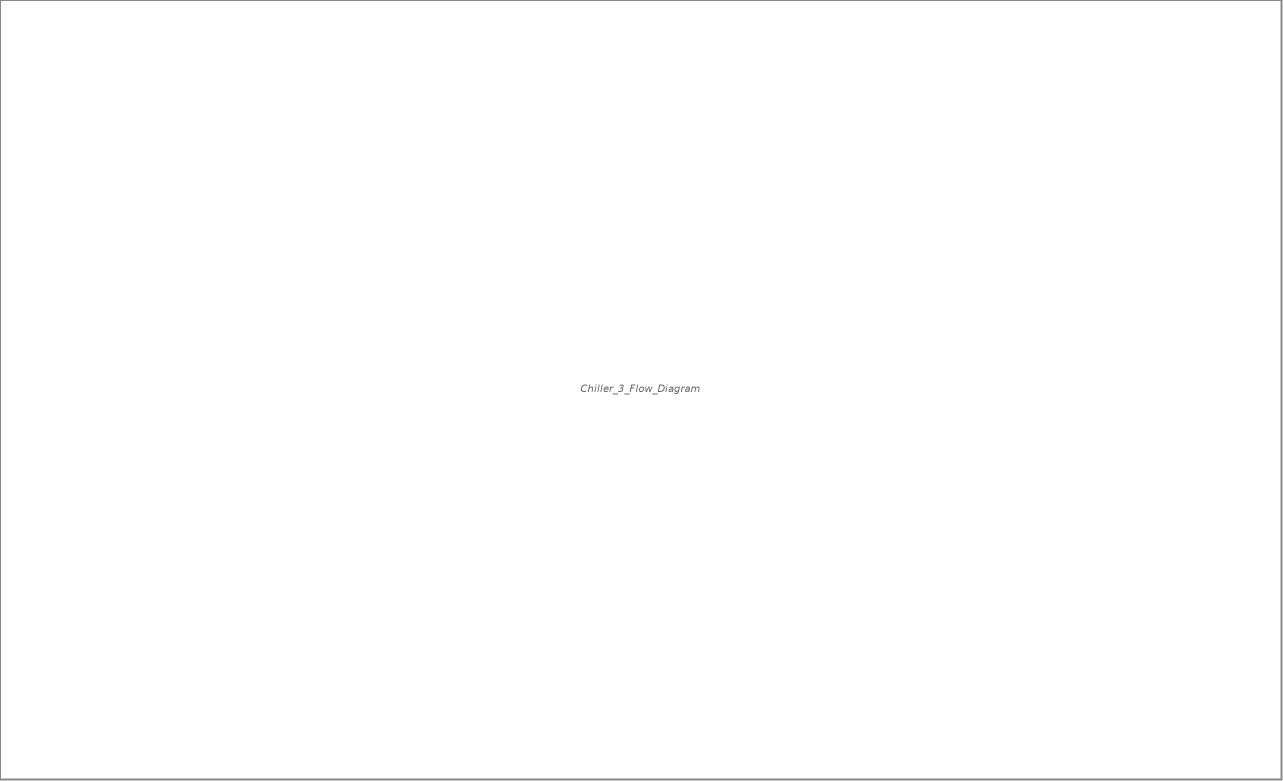
VISUALIZATION Chiller3Menu  // 1283x781
    TabControl (0,-2 1281x781)
        shows Chiller_3_Flow_Diagram()
        shows Chiller_3_Values()
        shows Chiller_3_Oil()
        shows Chiller_3_Alarm()
        shows Chiller_3_Trip()
        shows Chiller_3_VFD()
        [0]: TabTitle=Diagram
        [1]: TabTitle=Measured values
        [2]: TabTitle=Oil system
        [3]: TabTitle=Alarm
        [4]: TabTitle=Trip
END_VISUALIZATION

// /Chiller4Menu
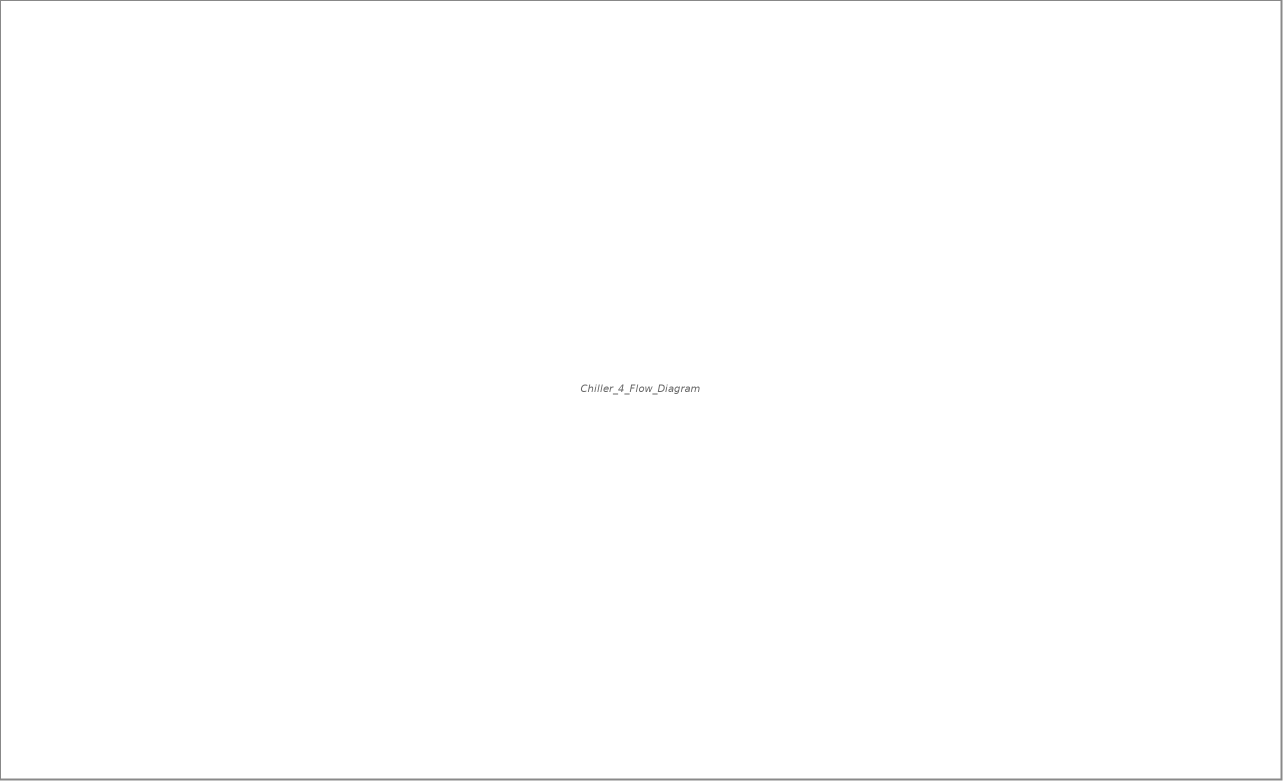
VISUALIZATION Chiller4Menu  // 1283x781
    TabControl (0,-2 1281x781)
        shows Chiller_4_Flow_Diagram()
        shows Chiller_4_Values()
        shows Chiller_4_Oil()
        shows Chiller_4_Alarm()
        shows Chiller_4_Trip()
        shows Chiller_4_VFD()
        [0]: TabTitle=Diagram
        [1]: TabTitle=Measured values
        [2]: TabTitle=Oil system
        [3]: TabTitle=Alarm
        [4]: TabTitle=Trip
END_VISUALIZATION

// /Chiller5Menu
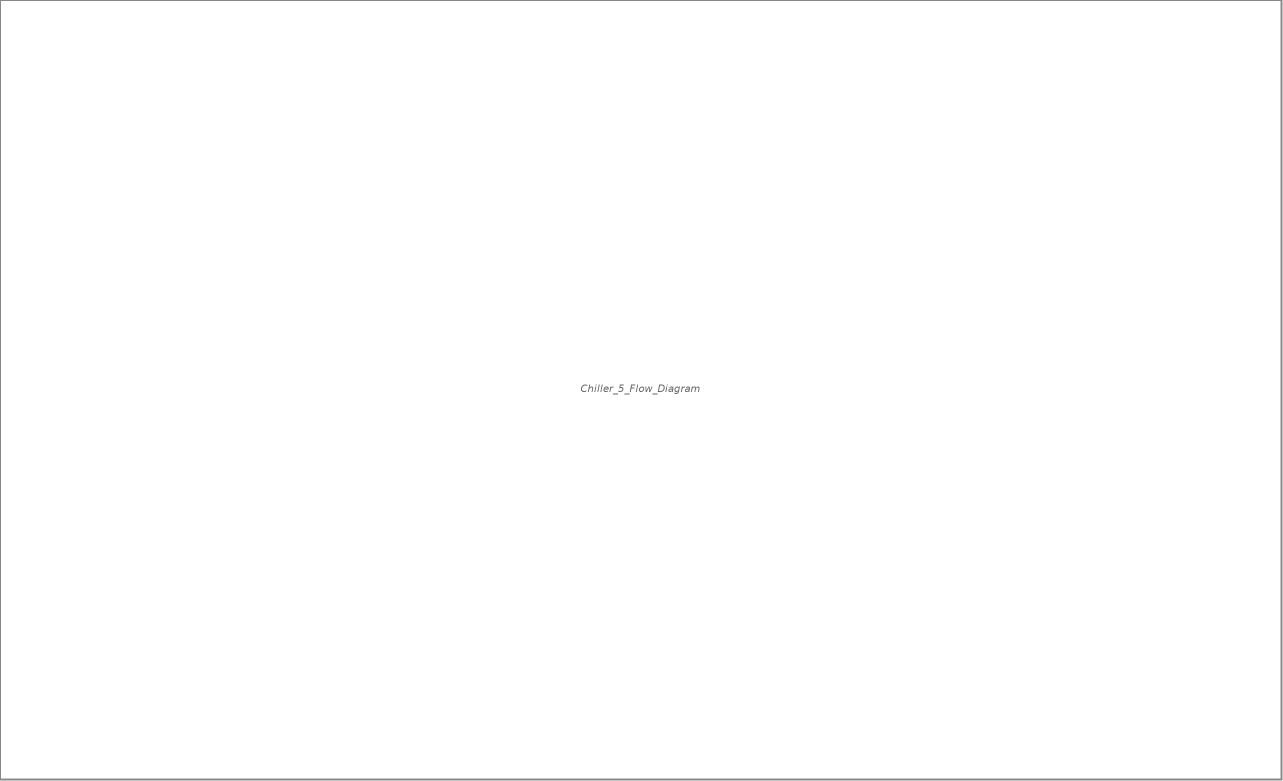
VISUALIZATION Chiller5Menu  // 1283x781
    TabControl (0,-2 1281x781)
        shows Chiller_5_Flow_Diagram()
        shows Chiller_5_Values()
        shows Chiller_5_Oil()
        shows Chiller_5_Alarm()
        shows Chiller_5_Trip()
        shows Chiller_4_VFD()
        [0]: TabTitle=Diagram
        [1]: TabTitle=Measured values
        [2]: TabTitle=Oil system
        [3]: TabTitle=Alarm
        [4]: TabTitle=Trip
END_VISUALIZATION

// /Chiller_1_Alarm
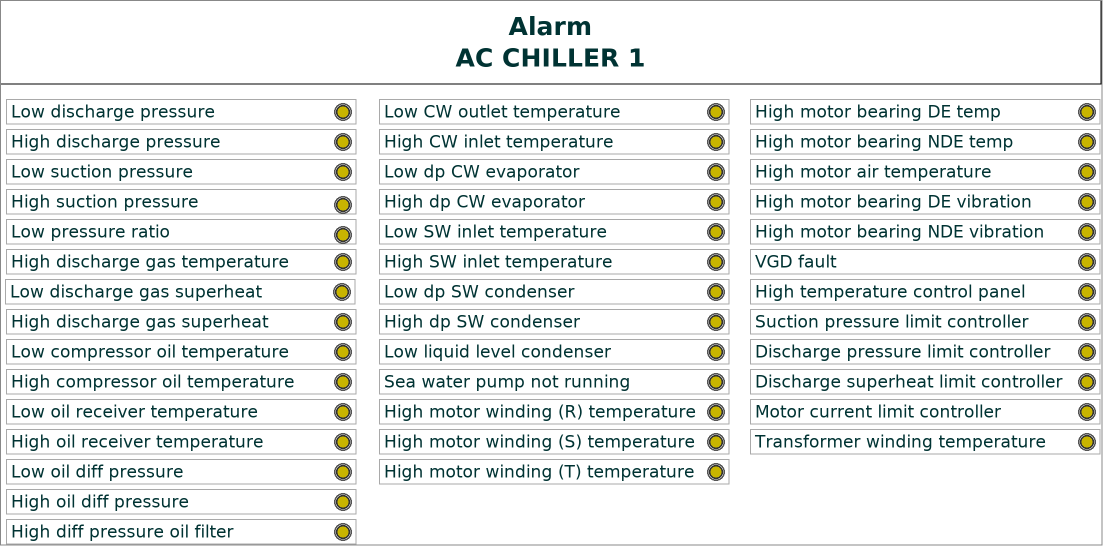
VISUALIZATION Chiller_1_Alarm  // 1103x546
    Rectangle (0,0 1101x84)
    Label (19,7 1063x70), "Alarm AC CHILLER 1"
    Rectangle (750,279 350x25)
    Label (752,281 316x21), "High temperature control panel"
    Lamp1 (1076,282 22x20), variable: Chiller_1.A_High_control_panel_temp, style: Lamp-Lamp1-Yellow
    Rectangle (750,309 350x25)
    Label (752,311 312x21), "Suction pressure limit controller"
    Lamp1 (1076,312 22x20), variable: Chiller_1.A_Suction_press_limit, style: Lamp-Lamp1-Yellow
    Rectangle (6,99 350x25)
    Label (8,101 318x21), "Low discharge pressure"
    Lamp1 (332,102 22x20), variable: Chiller_1.A_low_disch_press, style: Lamp-Lamp1-Yellow
    Rectangle (6,159 350x25)
    Label (8,161 319x21), "Low suction pressure"
    Lamp1 (332,162 22x20), variable: Chiller_1.A_Low_suction_pressure, style: Lamp-Lamp1-Yellow
    Rectangle (6,189 350x25)
    Label (8,191 322x21), "High suction pressure"
    Lamp1 (332,195 22x20), variable: Chiller_1.A_High_suction_pressure, style: Lamp-Lamp1-Yellow
    Rectangle (6,249 350x25)
    Label (8,251 317x21), "High discharge gas temperature"
    Lamp1 (332,252 22x20), variable: Chiller_1.A_High_discharge_temp, style: Lamp-Lamp1-Yellow
    Rectangle (379,399 350x25)
    Label (381,401 320x21), "High motor winding (R) temperature"
    Lamp1 (705,402 22x20), variable: Chiller_1.A_High_motor_wind_temp_R, style: Lamp-Lamp1-Yellow
    Rectangle (379,429 350x25)
    Label (381,431 319x21), "High motor winding (S) temperature"
    Lamp1 (705,432 22x20), variable: Chiller_1.A_High_motor_wind_temp_S, style: Lamp-Lamp1-Yellow
    Rectangle (6,369 350x25)
    Label (8,371 319x21), "High compressor oil temperature"
    Lamp1 (332,372 22x20), variable: Chiller_1.A_High_temp_oil_inlet_comp, style: Lamp-Lamp1-Yellow
    Rectangle (6,339 350x25)
    Label (8,341 322x21), "Low compressor oil temperature"
    Lamp1 (332,342 22x20), variable: Chiller_1.A_Low_temp_oil_inlet_comp, style: Lamp-Lamp1-Yellow
    Rectangle (6,429 350x25)
    Label (8,431 317x21), "High oil receiver temperature"
    Lamp1 (332,432 22x20), variable: Chiller_1.A_High_oil_temp_receiver, style: Lamp-Lamp1-Yellow
    Rectangle (6,399 350x25)
    Label (8,401 319x21), "Low oil receiver temperature"
    Lamp1 (332,402 22x20), variable: Chiller_1.A_Low_oil_temp_receiver, style: Lamp-Lamp1-Yellow
    Rectangle (6,459 350x25)
    Label (8,461 322x21), "Low oil diff pressure"
    Lamp1 (332,462 22x20), variable: Chiller_1.A_Low_oil_diff_pressure, style: Lamp-Lamp1-Yellow
    Rectangle (6,489 350x25)
    Label (8,491 317x21), "High oil diff pressure"
    Lamp1 (332,492 22x20), variable: Chiller_1.A_High_oil_diff_pressure, style: Lamp-Lamp1-Yellow
    Rectangle (6,309 350x25)
    Label (8,311 319x21), "High discharge gas superheat"
    Lamp1 (332,312 22x20), variable: Chiller_1.A_High_discharge_superheat, style: Lamp-Lamp1-Yellow
    Rectangle (5,279 350x25)
    Label (7,281 322x21), "Low discharge gas superheat"
    Lamp1 (331,282 22x20), variable: Chiller_1.A_Low_discharge_superheat, style: Lamp-Lamp1-Yellow
    Rectangle (379,219 350x25)
    Label (381,221 317x21), "Low SW inlet temperature"
    Lamp1 (705,222 22x20), variable: Chiller_1.A_Low_SW_inlet_temp, style: Lamp-Lamp1-Yellow
    Rectangle (379,129 350x25)
    Label (381,131 322x21), "High CW inlet temperature"
    Lamp1 (705,132 22x20), variable: Chiller_1.A_High_CW_inlet_temp, style: Lamp-Lamp1-Yellow
    Rectangle (379,99 350x25)
    Label (381,101 317x21), "Low CW outlet temperature"
    Lamp1 (705,102 22x20), variable: Chiller_1.A_Low_CW_outlet_temp, style: Lamp-Lamp1-Yellow
    Rectangle (6,519 350x25)
    Label (8,521 317x21), "High diff pressure oil filter"
    Lamp1 (332,522 22x20), variable: Chiller_1.A_High_oil_filter_diff_press, style: Lamp-Lamp1-Yellow
    Rectangle (379,459 350x25)
    Label (381,461 317x21), "High motor winding (T) temperature"
    Lamp1 (705,462 22x20), variable: Chiller_1.A_High_motor_wind_temp_T, style: Lamp-Lamp1-Yellow
    Rectangle (750,99 350x25)
    Label (752,101 317x21), "High motor bearing DE temp"
    Lamp1 (1076,102 22x20), variable: Chiller_1.A_High_comp_mo_DE_bear_temp, style: Lamp-Lamp1-Yellow
    Rectangle (750,129 350x25)
    Label (752,131 319x21), "High motor bearing NDE temp"
    Lamp1 (1076,132 22x20), variable: Chiller_1.A_High_comp_mo_NDE_bear_temp, style: Lamp-Lamp1-Yellow
    Rectangle (750,159 350x25)
    Label (752,161 322x21), "High motor air temperature"
    Lamp1 (1076,162 22x20), variable: Chiller_1.A_High_motor_air_temp, style: Lamp-Lamp1-Yellow
    Rectangle (750,189 350x25)
    Label (752,191 317x21), "High motor bearing DE vibration"
    Lamp1 (1076,192 22x20), variable: Chiller_1.A_High_comp_mo_DE_bear_vib, style: Lamp-Lamp1-Yellow
    Rectangle (750,219 350x25)
    Label (752,221 319x21), "High motor bearing NDE vibration"
    Lamp1 (1076,222 22x20), variable: Chiller_1.A_High_comp_mo_NDE_bear_vib, style: Lamp-Lamp1-Yellow
    Rectangle (379,189 350x25)
    Label (381,191 322x21), "High dp CW evaporator"
    Lamp1 (705,192 22x20), variable: Chiller_1.A_High_CW_dP, style: Lamp-Lamp1-Yellow
    Rectangle (379,159 350x25)
    Label (381,161 317x21), "Low dp CW evaporator"
    Lamp1 (705,162 22x20), variable: Chiller_1.A_Low_CW_dP, style: Lamp-Lamp1-Yellow
    Rectangle (379,309 350x25)
    Label (381,311 319x21), "High dp SW condenser"
    Lamp1 (705,312 22x20), variable: Chiller_1.A_High_SW_dP, style: Lamp-Lamp1-Yellow
    Rectangle (379,279 350x25)
    Label (381,281 322x21), "Low dp SW condenser"
    Lamp1 (705,282 22x20), variable: Chiller_1.A_Low_SW_dP, style: Lamp-Lamp1-Yellow
    Rectangle (750,249 350x25)
    Label (752,251 317x21), "VGD fault"
    Lamp1 (1076,252 22x20), variable: Chiller_1.A_VGD_Fault, style: Lamp-Lamp1-Yellow
    Rectangle (379,339 350x25)
    Label (381,341 317x21), "Low liquid level condenser"
    Lamp1 (705,342 22x20), variable: Chiller_1.A_Low_liquid_level, style: Lamp-Lamp1-Yellow
    Rectangle (6,129 350x25)
    Label (8,131 318x21), "High discharge pressure"
    Lamp1 (332,132 22x20), variable: Chiller_1.A_high_disch_press, style: Lamp-Lamp1-Yellow
    Rectangle (379,249 350x25)
    Label (381,251 314x21), "High SW inlet temperature"
    Lamp1 (705,252 22x20), variable: Chiller_1.A_High_SW_inlet_temp, style: Lamp-Lamp1-Yellow
    Rectangle (379,369 350x25)
    Label (381,371 314x21), "Sea water pump not running"
    Lamp1 (705,372 22x20), variable: Chiller_1.A_Seawater_pump_not_running, style: Lamp-Lamp1-Yellow
    Rectangle (750,339 350x25)
    Label (752,341 312x21), "Discharge pressure limit controller"
    Lamp1 (1076,342 22x20), variable: Chiller_1.A_Discharge_press_limit, style: Lamp-Lamp1-Yellow
    Rectangle (750,369 350x25)
    Label (752,371 312x21), "Discharge superheat limit controller"
    Lamp1 (1076,372 22x20), variable: Chiller_1.A_Discharge_superheat_limit, style: Lamp-Lamp1-Yellow
    Rectangle (750,399 350x25)
    Label (752,401 312x21), "Motor current limit controller"
    Lamp1 (1076,402 22x20), variable: Chiller_1.A_Motor_current_limit, style: Lamp-Lamp1-Yellow
    Rectangle (750,429 350x25)
    Label (752,431 312x21), "Transformer winding temperature"
    Lamp1 (1076,432 22x20), variable: Chiller_1.A_Transformer_winding_temp, style: Lamp-Lamp1-Yellow
    Rectangle (6,219 350x25)
    Label (8,221 322x21), "Low pressure ratio"
    Lamp1 (332,225 22x20), variable: Chiller_1.A_Low_press_ratio, style: Lamp-Lamp1-Yellow
END_VISUALIZATION

// /Chiller_1_Flow_Diagram
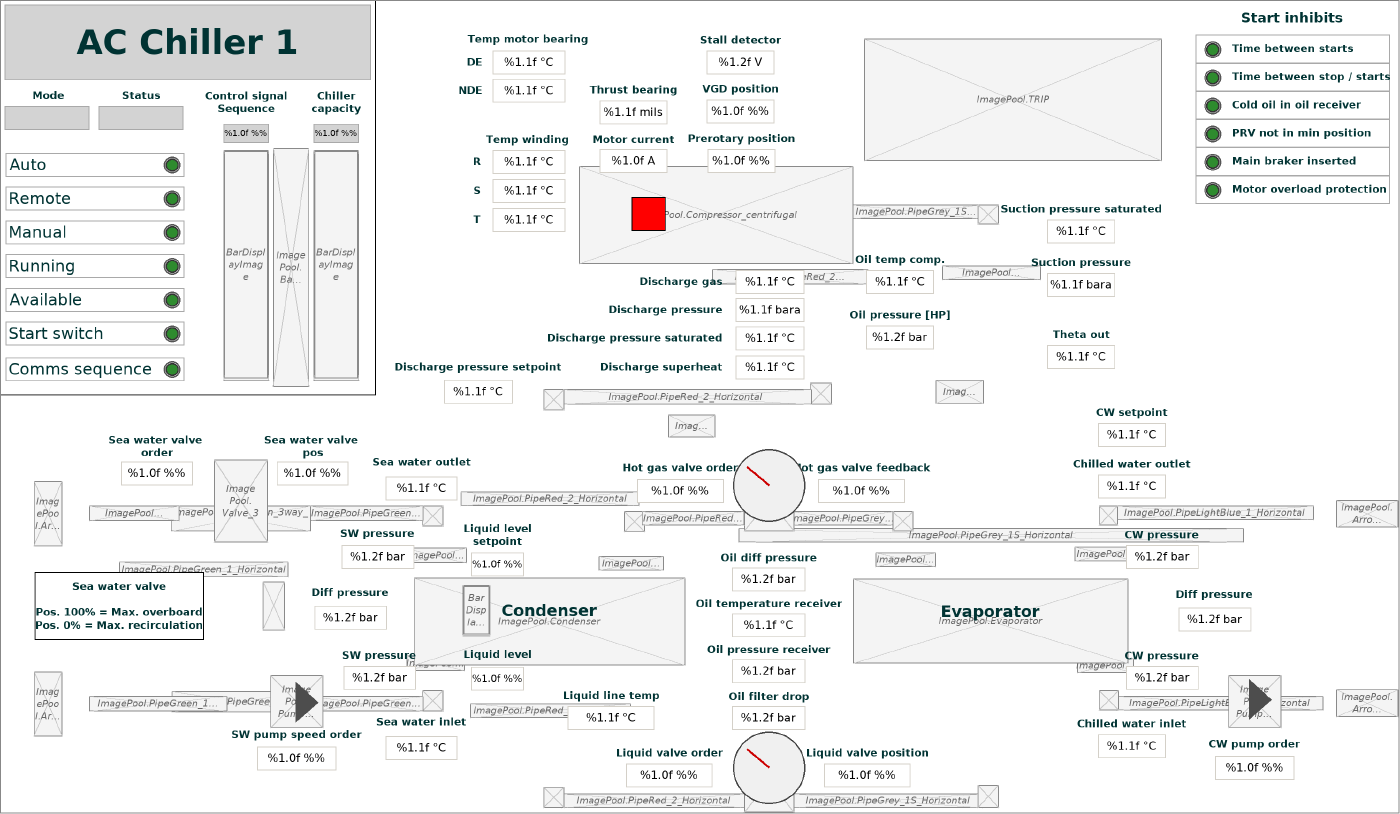
VISUALIZATION Chiller_1_Flow_Diagram  // 1492x868
    Rectangle (0,0 400x421)
    Textfield (238,132 48x20), "%1.0f %%", text variable: Sequence.Seq_cap_order_C1
        p4168582468: Sequence.Seq_cap_order_C1
    Image (1148,702 60x15), angle 270, image: ImagePool.PipeLightBlue_1_Horizontal
    Image (1145,583 67x15), angle 270, image: ImagePool.PipeLightBlue_1_Horizontal
    Image (908,218 137x15), image: ImagePool.PipeGrey_1S_Horizontal
    Image (845,846 202x15), image: ImagePool.PipeGrey_1S_Horizontal
    Image (933,589 64x15), angle 270, image: ImagePool.PipeGrey_1S_Horizontal
    Image (787,563 538x15), angle 270, image: ImagePool.PipeGrey_1S_Horizontal
    Image (843,545 110x15), image: ImagePool.PipeGrey_1S_Horizontal
    Image (638,593 69x15), angle 270, image: ImagePool.PipeRed_2_Horizontal
    Image (501,750 171x15), angle 270, image: ImagePool.PipeRed_2_Horizontal
    Label (218,94 89x30), "Control signal Sequence"
    Image (617,177 292x104), image: ImagePool.Compressor_centrifugal
    Image (759,287 166x16), angle 270, image: ImagePool.PipeRed_2_Horizontal
    Image (863,408 23x23), image: ImagePool.PipeRed_2_LU
    Image (596,415 269x16), image: ImagePool.PipeRed_2_Horizontal
    Image (909,617 293x90), image: ImagePool.Evaporator
    Image (431,584 66x16), angle 270, image: ImagePool.PipeGreen_1_Horizontal
    Image (450,539 22x22), image: ImagePool.PipeGreen_1_LD
    Image (329,539 122x16), image: ImagePool.PipeGreen_1_Horizontal
    Label (331,617 84x30), "Diff pressure"
    Textfield (335,646 77x25), "%1.2f bar", text variable: Chiller_1.dP_SW
        p4168582468: Chiller_1.dP_SW
    Image (127,599 180x16), angle 270, image: ImagePool.PipeGreen_1_Horizontal
    Image (183,737 147x22), image: ImagePool.PipeGreen_3way
    Image (433,699 62x16), angle 270, image: ImagePool.PipeGreen_1_Horizontal
    Image (450,736 22x22), image: ImagePool.PipeGreen_2_LU
    Image (329,742 122x16), image: ImagePool.PipeGreen_1_Horizontal
    Image (182,539 149x27), image: ImagePool.PipeGreen_3way_2
    Image (288,720 56x56), image: ImagePool.Pump_Large_3
    Polygon (315,746) (315,727) (339,749) (315,770) (315,762), colour toggle: Chiller_1.Sea_water_pump
    Image (36,513 30x69), angle 90, image: ImagePool.Arrow green down
    Image (36,716 30x69), angle 270, image: ImagePool.Arrow green down
    Image (579,415 22x22), image: ImagePool.PipeRed_1_RD
    Image (491,524 190x15), angle 270, image: ImagePool.PipeRed_2_Horizontal
    Label (360,554 84x30), "SW pressure"
    Textfield (364,581 77x25), "%1.2f bar", text variable: Chiller_1.Press_water_cond_out
        p4168582468: Chiller_1.Press_water_cond_out
    Image (95,539 96x16), image: ImagePool.PipeGreen_1_Horizontal
    Image (441,616 289x93), image: ImagePool.Condenser
    Image (598,846 197x15), image: ImagePool.PipeRed_2_Horizontal
    Image (579,839 22x22), image: ImagePool.PipeRed_2_RU
    Label (362,684 84x30), "SW pressure"
    Textfield (366,710 77x25), "%1.2f bar", text variable: Chiller_1.Press_water_cond_inlet
        p4168582468: Chiller_1.Press_water_cond_inlet
    Image (793,501 53x65), image: ImagePool.Valve_2
    Image (793,801 53x65), image: ImagePool.Valve_2
    Image (665,545 22x22), image: ImagePool.PipeRed_1_RD
    Image (684,545 109x15), image: ImagePool.PipeRed_2_Horizontal
    Image (951,545 22x21), image: ImagePool.PipeGrey_2_LD
    Image (1042,837 22x24), image: ImagePool.PipeGrey_3_LU
    Image (1042,218 22x21), image: ImagePool.PipeGrey_2_LD
    Image (1004,283 105x15), angle 270, image: ImagePool.PipeGrey_1S_Horizontal
    Label (521,636 129x30), "Condenser"
    Label (991,637 129x30), "Evaporator"
    Image (1189,539 211x15), image: ImagePool.PipeLightBlue_1_Horizontal
    Image (1171,539 20x21), image: ImagePool.PipeLightBlue_3_RD
    Image (1190,742 220x15), image: ImagePool.PipeLightBlue_1_Horizontal
    Image (1171,736 21x21), image: ImagePool.PipeLightBlue_3_RU
    Image (1424,533 66x29), angle 180, image: ImagePool.Arrow lightblue left
    Image (1424,735 66x29), image: ImagePool.Arrow lightblue left
    Image (1309,720 56x56), image: ImagePool.Pump_Large_3
    Polygon (1331,743) (1331,724) (1355,746) (1331,767) (1331,759), colour toggle: Chiller_1.CW_Flow_ind
    Image (280,620 23x52), image: ImagePool.Arrow green down
    Image (712,442 50x24), image: ImagePool.Arrow red left
    Image (997,405 51x25), angle 90, image: ImagePool.Arrow gray left
    Image (291,158 38x254), image: ImagePool.BarScale3
    Label (324,94 69x30), "Chiller capacity"
    Textfield (105,113 90x25), text list: 'TextList_PT', text index: Chiller_1.Unit_switch_status
    Textfield (5,113 90x25), text list: 'TextList_PT', text index: Chiller_1.Unit_start_switch
    Textfield (334,132 48x20), "%1.0f %%", text variable: Chiller_1.Chiller_capacity_t1
        p4168582468: Chiller_1.Chiller_capacity_t1
    Textfield (5,5 390x80), "AC Chiller 1"
    Textfield (525,160 77x25), "%1.1f °C", text variable: Chiller_1.Temp_motor_wind_R
        p4168582468: Chiller_1.Temp_motor_wind_R
    Label (496,160 25x25), "R"
    Textfield (525,191 77x25), "%1.1f °C", text variable: Chiller_1.Temp_motor_wind_S
        p4168582468: Chiller_1.Temp_motor_wind_S
    Label (496,191 25x25), "S"
    Textfield (525,222 77x25), "%1.1f °C", text variable: Chiller_1.Temp_motor_wind_T
        p4168582468: Chiller_1.Temp_motor_wind_T
    Label (496,222 25x25), "T"
    Textfield (679,511 92x25), "%1.0f %%", text variable: Chiller_1.Hot_gas_valve_output
        p4168582468: Chiller_1.Hot_gas_valve_output
    Label (664,484 122x30), "Hot gas valve order"
    Label (849,484 139x30), "Hot gas valve feedback"
    Textfield (872,511 92x25), "%1.0f %%", text variable: Chiller_1.Feedback_HGV
        p4168582468: Chiller_1.Feedback_HGV
    Meter360 (781,479 77x77), value: Chiller_1.Feedback_HGV, style: Meter-Meter360-Gray, scale format: %1.0f, scale 0..100
        p3451962224: ImagePool.Invisible
    Meter360 (781,780 77x77), value: Chiller_1.Feedback_liquid_valve, style: Meter-Meter360-Gray, scale format: %1.0f, scale 0..100
        p3451962224: ImagePool.Invisible
    Textfield (502,589 56x25), "%1.0f %%", text variable: Chiller_1.SP_PID_Level
        p4168582468: Chiller_1.SP_PID_Level
    Label (494,551 73x39), "Liquid level setpoint"
    Textfield (502,711 56x25), "%1.0f %%", text variable: Chiller_1.Liquid_level_condenser
        p4168582468: Chiller_1.Liquid_level_condenser
    Label (491,683 79x30), "Liquid level"
    Textfield (639,159 72x25), "%1.0f A", text variable: Chiller_1.Motor_current
        p4168582468: Chiller_1.Motor_current
    Label (634,138 83x22), "Motor current"
    Textfield (274,796 84x25), "%1.0f %%", text variable: Chiller_1.SW_pump_speed_order
        p4168582468: Chiller_1.SW_pump_speed_order
    Label (250,770 132x27), "SW pump speed order"
    Textfield (473,405 73x25), "%1.1f °C", tooltip "Chiller_1.SP_cond_press", text variable: Chiller_1.SP_cond_press
        p4168582468: Chiller_1.SP_cond_press
    Textfield (784,348 73x25), "%1.1f °C", text variable: Chiller_1.Discharge_saturated_temp
        p4168582468: Chiller_1.Discharge_saturated_temp
    Label (589,347 184x27), "Discharge pressure saturated"
    Label (425,378 169x27), "Discharge pressure setpoint"
    Textfield (411,785 76x25), "%1.1f °C", text variable: Chiller_1.Temp_water_inlet_cond
        p4168582468: Chiller_1.Temp_water_inlet_cond
    Label (399,755 100x30), "Sea water inlet"
    Textfield (411,508 76x25), "%1.1f °C", text variable: Chiller_1.Temp_water_outlet_cond
        p4168582468: Chiller_1.Temp_water_outlet_cond
    Label (397,478 105x30), "Sea water outlet"
    Label (500,27 126x30), "Temp motor bearing"
    Textfield (525,84 77x25), "%1.1f °C", text variable: Chiller_1.Temp_motor_bearing_NDE
        p4168582468: Chiller_1.Temp_motor_bearing_NDE
    Textfield (525,54 77x25), "%1.1f °C", text variable: Chiller_1.Temp_motor_bearing_DE
        p4168582468: Chiller_1.Temp_motor_bearing_DE
    Label (480,54 37x25), "DE"
    Label (480,84 37x25), "NDE"
    Label (678,287 95x27), "Discharge gas"
    Textfield (784,288 73x25), "%1.1f °C", text variable: Chiller_1.Temp_discharge
        p4168582468: Chiller_1.Temp_discharge
    Label (644,317 129x27), "Discharge pressure"
    Textfield (784,318 73x25), "%1.1f bara", text variable: Chiller_1.Press_discharge_compr
        p4168582468: Chiller_1.Press_discharge_compr
    Textfield (784,379 73x25), "%1.1f °C", text variable: Chiller_1.Discharge_superheat
        p4168582468: Chiller_1.Discharge_superheat
    Label (589,378 184x27), "Discharge superheat"
    Label (631,84 89x24), "Thrust bearing"
    Textfield (639,107 72x25), "%1.1f mils", text variable: Chiller_1.Thrust_bearing_position
        p4168582468: Chiller_1.Thrust_bearing_position
    Label (857,788 135x30), "Liquid valve position"
    Textfield (878,814 92x25), "%1.0f %%", text variable: Chiller_1.Feedback_liquid_valve
        p4168582468: Chiller_1.Feedback_liquid_valve
    Textfield (780,753 78x25), "%1.2f bar", text variable: Chiller_1.Oil_Filter_Drop
        p4168582468: Chiller_1.Oil_Filter_Drop
    Label (778,732 83x22), "Oil filter drop"
    Textfield (667,814 92x25), "%1.0f %%", text variable: Chiller_1.Liquid_valve_output
        p4168582468: Chiller_1.Liquid_valve_output
    Label (646,788 135x30), "Liquid valve order"
    Textfield (780,703 78x25), "%1.2f bar", text variable: Chiller_1.Press_oil_receiver
        p4168582468: Chiller_1.Press_oil_receiver
    Label (752,682 135x22), "Oil pressure receiver"
    Textfield (780,654 78x25), "%1.1f °C", text variable: Chiller_1.Oil_temp_receiver
        p4168582468: Chiller_1.Oil_temp_receiver
    Label (748,633 143x22), "Oil temperature receiver"
    Textfield (780,605 78x25), "%1.2f bar", text variable: Chiller_1.Oil_diff_pressure
        p4168582468: Chiller_1.Oil_diff_pressure
    Label (769,584 101x22), "Oil diff pressure"
    Label (736,136 109x24), "Prerotary position"
    Textfield (754,159 72x25), "%1.0f %%", text variable: Chiller_1.Feedback_PRV
        p4168582468: Chiller_1.Feedback_PRV
    Label (746,83 87x24), "VGD position"
    Textfield (753,106 72x25), "%1.0f %%", text variable: Chiller_1.Feedback_VGD
        p4168582468: Chiller_1.Feedback_VGD
    Label (746,31 87x24), "Stall detector"
    Textfield (753,54 72x25), "%1.2f V", text variable: Chiller_1.Stall_detector
        p4168582468: Chiller_1.Stall_detector
    Label (1067,211 171x24), "Suction pressure saturated"
    Textfield (1116,234 72x25), "%1.1f °C", text variable: Chiller_1.Suction_saturated_temp
        p4168582468: Chiller_1.Suction_saturated_temp
    Textfield (1116,291 72x25), "%1.1f bara", text variable: Chiller_1.Press_suction_compr
        p4168582468: Chiller_1.Press_suction_compr
    Label (1067,268 171x24), "Suction pressure"
    Textfield (1116,368 72x25), "%1.1f °C", text variable: Chiller_1.Theta_out
        p4168582468: Chiller_1.Theta_out
    Label (1111,345 83x24), "Theta out"
    Label (1196,557 84x27), "CW pressure"
    Textfield (1200,581 77x25), "%1.2f bar", text variable: Chiller_1.Press_chilled_medium_out
        p4168582468: Chiller_1.Press_chilled_medium_out
    Textfield (1200,710 77x25), "%1.2f bar", text variable: Chiller_1.Press_chilled_medium_in
        p4168582468: Chiller_1.Press_chilled_medium_in
    Label (1196,686 84x27), "CW pressure"
    Textfield (1170,506 72x25), "%1.1f °C", text variable: Chiller_1.Temp_chilled_medium_out
        p4168582468: Chiller_1.Temp_chilled_medium_out
    Label (1146,483 121x24), "Chilled water outlet"
    Label (1146,428 121x24), "CW setpoint"
    Textfield (1170,451 72x25), "%1.1f °C", text variable: Chiller_1.SP_CW_controller
        p4168582468: Chiller_1.SP_CW_controller
    Label (1252,619 84x30), "Diff pressure"
    Textfield (1256,648 77x25), "%1.2f bar", text variable: Chiller_1.dP_CW
        p4168582468: Chiller_1.dP_CW
    Textfield (1170,783 72x25), "%1.1f °C", text variable: Chiller_1.Temp_chilled_medium_in
        p4168582468: Chiller_1.Temp_chilled_medium_in
    Label (1146,760 121x24), "Chilled water inlet"
    Group (6,271 190x25)
        Rectangle (0,0 190x25)
        Label (0,2 105x21), "Running"
        Lamp1 (166,3 23x20), variable: Chiller_1.Unit_running, style: Lamp-Lamp1-Green
    Group (6,163 190x25)
        Rectangle (0,0 190x25)
        Label (1,2 105x21), "Auto"
        Lamp1 (166,3 23x20), variable: Chiller_1.Unit_auto, style: Lamp-Lamp1-Green
    Group (6,199 190x25)
        Rectangle (0,0 190x25)
        Label (0,2 105x21), "Remote"
        Lamp1 (166,3 23x20), variable: Chiller_1.Unit_remote, style: Lamp-Lamp1-Green
    Group (6,235 190x25)
        Rectangle (0,0 190x25)
        Label (0,2 105x21), "Manual"
        Lamp1 (166,3 23x20), variable: Chiller_1.Unit_manual, style: Lamp-Lamp1-Green
    Group (6,307 190x25)
        Rectangle (0,0 190x25)
        Label (1,2 105x21), "Available"
        Lamp1 (166,3 23x20), variable: Chiller_1.Unit_available, style: Lamp-Lamp1-Green
    Group (6,343 190x25)
        Rectangle (0,0 190x25)
        Label (0,2 130x21), "Start switch"
        Lamp1 (166,3 23x20), variable: Chiller_1.Unit_start_switch, style: Lamp-Lamp1-Green
    Group (6,381 190x25)
        Rectangle (0,0 190x25)
        Label (0,2 160x21), "Comms sequence"
        Lamp1 (166,3 23x20), variable: not.Sequence.A_Comms_chiller_1, style: Lamp-Lamp1-Green
    Label (912,265 95x24), "Oil temp comp."
    Textfield (923,288 72x25), "%1.1f °C", text variable: Chiller_1.Temp_oil_inlet_compr
        p4168582468: Chiller_1.Temp_oil_inlet_compr
    Label (902,324 115x24), "Oil pressure [HP]"
    Textfield (923,347 72x25), "%1.2f bar", text variable: Chiller_1.Press_oil_compr
        p4168582468: Chiller_1.Press_oil_compr
    Image (921,41 317x130), invisible if: Chiller_1.Unit_alarm, image: ImagePool.ALARM
    Image (921,41 317x130), invisible if: Chiller_1.Unit_trip, image: ImagePool.TRIP
    Label (7,87 89x30), "Mode"
    Label (106,87 89x30), "Status"
    Rectangle (334,160 48x246)
    Image (238,160 48x246), image: ImagePool.CapBarTranparant
    BarDisplayImage (239,161 46x242), value: Sequence.Seq_cap_order_C1, style: BarDisplayImage-Gray, scale format: %.0f, scale 0..100
        p3451962224: ImagePool.Invisible
    Rectangle (673,210 36x36), colour toggle: Chiller_1.Unit_running
    Rectangle (673,210 36x36), colour toggle: Chiller_1.Unit_alarm
    Rectangle (673,210 36x36), colour toggle: Chiller_1.Unit_trip
    Image (334,160 48x246), image: ImagePool.CapBarTranparant
    BarDisplayImage (335,161 46x242), value: Chiller_1.Chiller_capacity_t1, style: BarDisplayImage-Gray, scale format: %.0f, scale 0..100
        p3451962224: ImagePool.Invisible
    Rectangle (493,624 28x52)
    Image (493,624 29x54), image: ImagePool.CapBarTranparant
    BarDisplayImage (494,625 27x51), value: Chiller_1.Liquid_level_condenser, style: BarDisplayImage-Gray, scale format: %.0f, scale 0..100
        p3451962224: ImagePool.Invisible
    Image (95,742 147x16), image: ImagePool.PipeGreen_1_Horizontal
    Textfield (605,753 92x25), "%1.1f °C", text variable: Chiller_1.Liquid_line_temp
        p4168582468: Chiller_1.Liquid_line_temp
    Label (595,727 113x30), "Liquid line temp"
    Image (228,490 57x88), image: ImagePool.Valve_3
    Label (115,461 105x30), "Sea water valve order"
    Textfield (129,492 76x25), "%1.0f %%", text variable: Chiller_1.Order_SWW_overboard
        p4168582468: Chiller_1.Order_SWW_overboard
    Label (281,461 105x30), "Sea water valve pos"
    Textfield (295,492 76x25), "%1.0f %%", text variable: Chiller_1.Feedback_seawater_valve_overboard
        p4168582468: Chiller_1.Feedback_seawater_valve_overboard
    Group (37,610 180x72)
        Rectangle (0,0 180x72)
        Label (0,0 180x72), "Sea water valve Pos. 100% = Max. overboard Pos. 0% = Max. recirculation"
    Label (511,138 103x22), "Temp winding"
    Rectangle (1274,37 207x30)
    Label (1310,38 142x28), "Time between starts"
    Lamp1 (1281,43 23x20), variable: Chiller_1.Start_inhib_time_between_Start, style: Lamp-Lamp1-Green
    Rectangle (1274,67 207x30)
    Label (1310,68 162x28), "Time between stop / starts"
    Lamp1 (1281,73 23x20), variable: Chiller_1.Start_inhib_time_between_Stop_Start, style: Lamp-Lamp1-Green
    Label (1307,7 140x24), "Start inhibits"
    Rectangle (1274,97 207x30)
    Label (1310,98 162x28), "Cold oil in oil receiver"
    Lamp1 (1281,103 23x20), variable: Chiller_1.Start_inhib_time_Oil_receiver_temp, style: Lamp-Lamp1-Green
    Rectangle (1274,127 207x30)
    Label (1310,128 162x28), "PRV not in min position"
    Lamp1 (1281,133 23x20), variable: Chiller_1.Start_inhib_PRV_not_min, style: Lamp-Lamp1-Green
    Rectangle (1274,157 207x30)
    Label (1310,158 162x28), "Main braker inserted"
    Lamp1 (1281,163 23x20), variable: not.Chiller_1.DO_9_0_Main_breaker_ready, style: Lamp-Lamp1-Green
    Textfield (1295,806 84x25), "%1.0f %%", text variable: Chiller_1.CW_Pump_Speed_SP
        p4168582468: Chiller_1.CW_Pump_Speed_SP
    Label (1271,780 132x27), "CW pump order"
    Rectangle (1274,187 207x30)
    Label (1310,188 162x28), "Motor overload protection"
    Lamp1 (1281,193 23x20), variable: not.Chiller_1.DI_0_6_Overload_protection, style: Lamp-Lamp1-Green
END_VISUALIZATION

// /Chiller_1_Oil
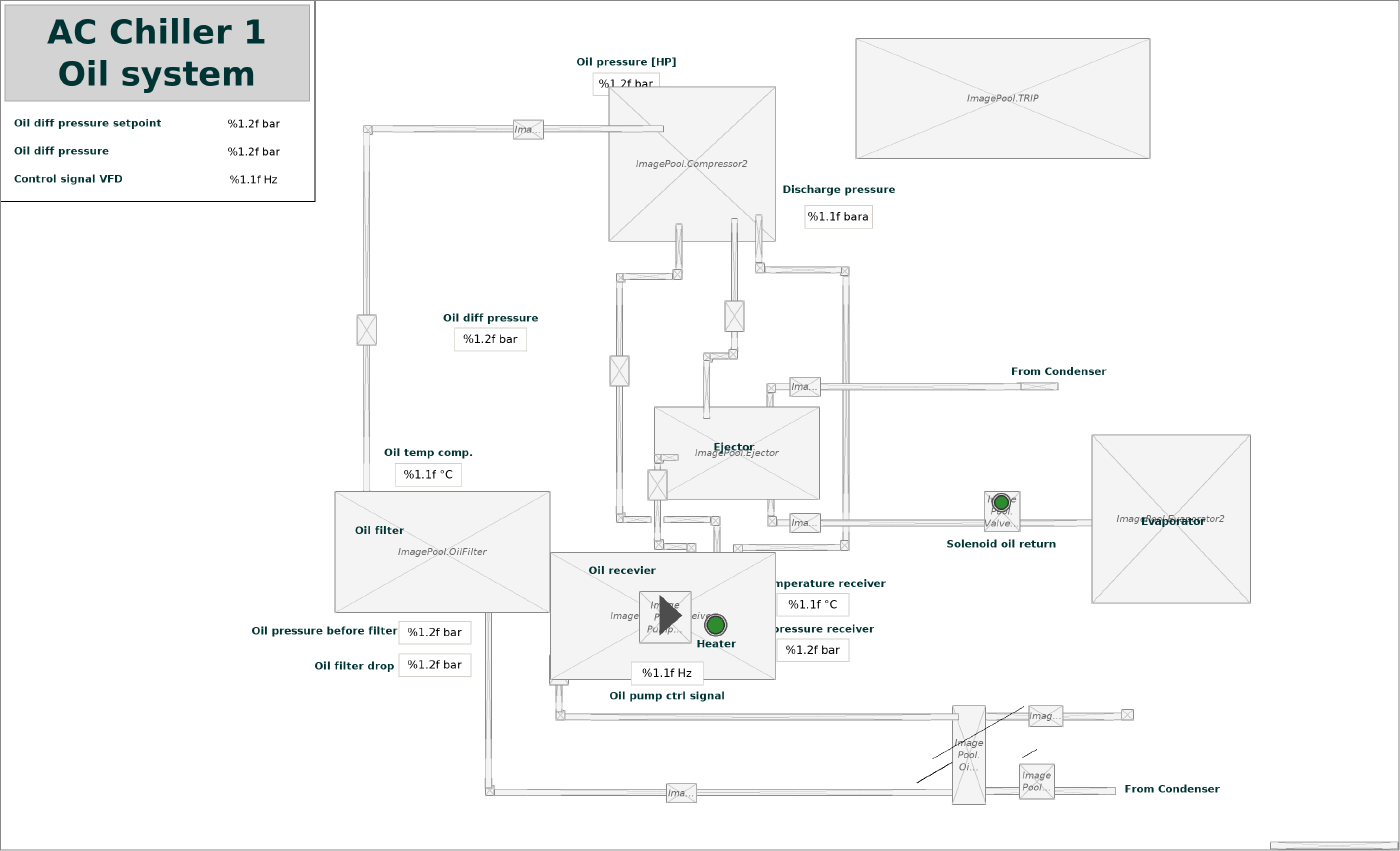
VISUALIZATION Chiller_1_Oil  // 1507x917
    Image (1094,412 45x8), angle 180, image: ImagePool.PipeBlack_1S_H_Faded
    Rectangle (0,0 339x217)
    Image (1367,907 138x8), angle 270, image: ImagePool.PipeGrey_1S_Horizontal
    Image (1053,768 155x8), image: ImagePool.PipeGrey_1S_Horizontal
    Image (1207,764 13x12), image: ImagePool.PipeGrey_3_LU
    Textfield (5,5 328x104), "AC Chiller 1 Oil system"
    Label (1066,387 128x27), "From Condenser"
    Label (838,191 129x27), "Discharge pressure"
    Textfield (866,221 73x25), "%1.1f bara", text variable: Chiller_1.Press_discharge_compr
        p4168582468: Chiller_1.Press_discharge_compr
    Label (1007,573 142x27), "Solenoid oil return"
    Textfield (429,704 78x25), "%1.2f bar", text variable: Chiller_1.Oil_Filter_Drop
        p4168582468: Chiller_1.Oil_Filter_Drop
    Label (340,707 83x22), "Oil filter drop"
    Textfield (836,688 78x25), "%1.2f bar", text variable: Chiller_1.Press_oil_receiver
        p4168582468: Chiller_1.Press_oil_receiver
    Label (808,667 135x22), "Oil pressure receiver"
    Textfield (836,639 78x25), "%1.1f °C", text variable: Chiller_1.Oil_temp_receiver
        p4168582468: Chiller_1.Oil_temp_receiver
    Label (804,618 143x22), "Oil temperature receiver"
    Textfield (489,353 78x25), "%1.2f bar", text variable: Chiller_1.Oil_diff_pressure
        p4168582468: Chiller_1.Oil_diff_pressure
    Label (478,332 101x22), "Oil diff pressure"
    Label (414,476 95x24), "Oil temp comp."
    Textfield (425,499 72x25), "%1.1f °C", text variable: Chiller_1.Temp_oil_inlet_compr
        p4168582468: Chiller_1.Temp_oil_inlet_compr
    Label (617,55 115x24), "Oil pressure [HP]"
    Textfield (638,78 72x25), "%1.2f bar", text variable: Chiller_1.Press_oil_compr
        p4168582468: Chiller_1.Press_oil_compr
    Image (921,41 317x130), invisible if: Chiller_1.Unit_alarm, image: ImagePool.ALARM
    Image (921,41 317x130), invisible if: Chiller_1.Unit_trip, image: ImagePool.TRIP
    Textfield (238,122 70x23), "%1.2f bar", text variable: Chiller_1.SP_oil_pressure
    Label (12,118 193x30), "Oil diff pressure setpoint"
    Textfield (238,152 70x23), "%1.2f bar", text variable: Chiller_1.Oil_diff_pressure
    Label (12,148 193x30), "Oil diff pressure"
    Textfield (238,182 70x23), "%1.1f Hz", text variable: Chiller_1.Setpoint_conv_oil_pump
    Label (12,178 131x30), "Control signal VFD"
    Label (651,739 135x22), "Oil pump ctrl signal"
    Textfield (429,669 78x25), "%1.2f bar", text variable: Chiller_1.Oil_pressure_before_filter
        p4168582468: Chiller_1.Oil_pressure_before_filter
    Label (276,669 147x22), "Oil pressure before filter"
    Label (1210,837 106x27), "From Condenser"
    Image (655,93 180x167), image: ImagePool.Compressor2
    Image (1051,848 150x8), angle 180, image: ImagePool.PipeBlack_1S_H_Faded
    Image (798,586 108x7), image: ImagePool.PipeBlack_1_Horizontal
    Image (907,297 7x286), image: ImagePool.PipeBlack_1_Vertical
    Image (391,135 10x10), image: ImagePool.PipeBlack_1_RD
    Image (522,846 10x11), image: ImagePool.PipeBlack_1_RU
    Image (1107,760 37x23), image: ImagePool.Arrow gray right
    Image (836,560 348x7), image: ImagePool.PipeBlack_1_Horizontal
    Image (1175,468 171x182), image: ImagePool.Evaporator2
    Image (826,512 7x44), image: ImagePool.PipeBlack_1_Vertical
    Image (826,556 10x11), image: ImagePool.PipeBlack_1_RU
    Image (789,596 7x28), image: ImagePool.PipeBlack_1_Vertical
    Image (789,586 10x10), image: ImagePool.PipeBlack_1_RD
    Image (904,582 10x11), image: ImagePool.PipeBlack_1_LU
    Image (850,553 33x21), image: ImagePool.Arrow black left
    Image (904,287 10x10), image: ImagePool.PipeBlack_1_LD
    Image (823,287 83x7), image: ImagePool.PipeBlack_1_Horizontal
    Image (813,283 10x11), image: ImagePool.PipeBlack_1_RU
    Image (813,231 7x52), image: ImagePool.PipeBlack_1_Vertical
    Image (825,413 10x10), image: ImagePool.PipeBlack_1_RD
    Image (834,413 265x7), image: ImagePool.PipeBlack_1_Horizontal
    Image (825,423 7x28), image: ImagePool.PipeBlack_1_Vertical
    Image (704,438 178x100), image: ImagePool.Ejector
    Image (850,406 33x21), image: ImagePool.Arrow black left
    Image (532,850 500x7), image: ImagePool.PipeBlack_1_Horizontal
    Image (1025,760 36x107), image: ImagePool.OilHeatExchanger
    Image (605,769 427x7), image: ImagePool.PipeBlack_1_Horizontal
    Image (598,765 10x11), image: ImagePool.PipeBlack_1_RU
    Image (598,670 7x97), image: ImagePool.PipeBlack_1_Vertical
    Image (598,660 10x10), image: ImagePool.PipeBlack_1_RD
    Image (605,660 19x7), image: ImagePool.PipeBlack_1_Horizontal
    Image (591,705 21x33), image: ImagePool.Arrow black down
    Image (717,844 33x21), image: ImagePool.Arrow black left
    Image (768,566 7x50), image: ImagePool.PipeBlack_1_Vertical
    Image (765,556 10x10), image: ImagePool.PipeBlack_1_LD
    Image (714,556 51x7), image: ImagePool.PipeBlack_1_Horizontal
    Image (704,581 10x11), image: ImagePool.PipeBlack_1_RU
    Image (704,499 7x84), image: ImagePool.PipeBlack_1_Vertical
    Image (704,489 10x10), image: ImagePool.PipeBlack_1_RD
    Image (711,489 19x7), image: ImagePool.PipeBlack_1_Horizontal
    Image (697,506 21x33), image: ImagePool.Arrow black down
    Image (714,585 28x7), image: ImagePool.PipeBlack_1_Horizontal
    Image (739,585 10x10), image: ImagePool.PipeBlack_1_LD
    Image (742,595 7x21), image: ImagePool.PipeBlack_1_Vertical
    Image (592,595 243x137), image: ImagePool.OilReceiver
    Image (400,135 314x7), image: ImagePool.PipeBlack_1_Horizontal
    Label (630,604 80x22), "Oil recevier"
    Image (522,553 7x296), image: ImagePool.PipeBlack_1_Vertical
    Image (519,544 10x10), image: ImagePool.PipeBlack_1_LD
    Image (400,544 120x7), image: ImagePool.PipeBlack_1_Horizontal
    Image (391,540 10x11), image: ImagePool.PipeBlack_1_RU
    Image (391,142 7x400), image: ImagePool.PipeBlack_1_Vertical
    Image (663,552 10x11), image: ImagePool.PipeBlack_1_RU
    Image (663,301 7x253), image: ImagePool.PipeBlack_1_Vertical
    Image (663,294 10x10), image: ImagePool.PipeBlack_1_RD
    Image (670,294 54x7), image: ImagePool.PipeBlack_1_Horizontal
    Image (656,383 21x33), image: ImagePool.Arrow black down
    Image (670,556 31x7), image: ImagePool.PipeBlack_1_Horizontal
    Image (727,241 7x53), image: ImagePool.PipeBlack_1_Vertical
    Image (724,290 10x11), image: ImagePool.PipeBlack_1_LU
    Image (757,380 10x10), image: ImagePool.PipeBlack_1_RD
    Image (764,380 22x7), image: ImagePool.PipeBlack_1_Horizontal
    Image (787,235 7x144), image: ImagePool.PipeBlack_1_Vertical
    Image (784,376 10x11), image: ImagePool.PipeBlack_1_LU
    Image (757,388 7x63), image: ImagePool.PipeBlack_1_Vertical
    Image (780,324 21x33), image: ImagePool.Arrow black down
    Label (750,471 80x22), "Ejector"
    Label (1223,551 80x22), "Evaporator"
    Image (384,339 21x33), image: ImagePool.Arrow black up
    Image (552,129 33x21), image: ImagePool.Arrow black right
    Image (360,529 232x131), image: ImagePool.OilFilter
    Label (379,561 59x22), "Oil filter"
    Line (987,843) (1025,821)
    Line (1100,816) (1116,807)
    Line (1004,817) (1102,761)
    Image (1097,823 38x38), image: ImagePool.RegValve
    Image (688,637 56x56), image: ImagePool.Pump_Large_3
    Polygon (710,660) (710,641) (734,663) (710,684) (710,676), colour toggle: Chiller_1.Comp_oil_pump
    Lamp1 (756,656 29x35), variable: Chiller_1.DO_0_6_Oil_heater, style: Lamp-Lamp1-Green
    Label (744,683 55x22), "Heater"
    Image (1059,529 39x44), image: ImagePool.Valve_2
    Lamp1 (1066,529 24x25), variable: Chiller_1.DO_0_4_Solenoid_valve_oil, style: Lamp-Lamp1-Green
    Textfield (679,713 78x25), "%1.1f Hz", text variable: Chiller_1.Setpoint_conv_oil_pump
END_VISUALIZATION

// /Chiller_1_Trip
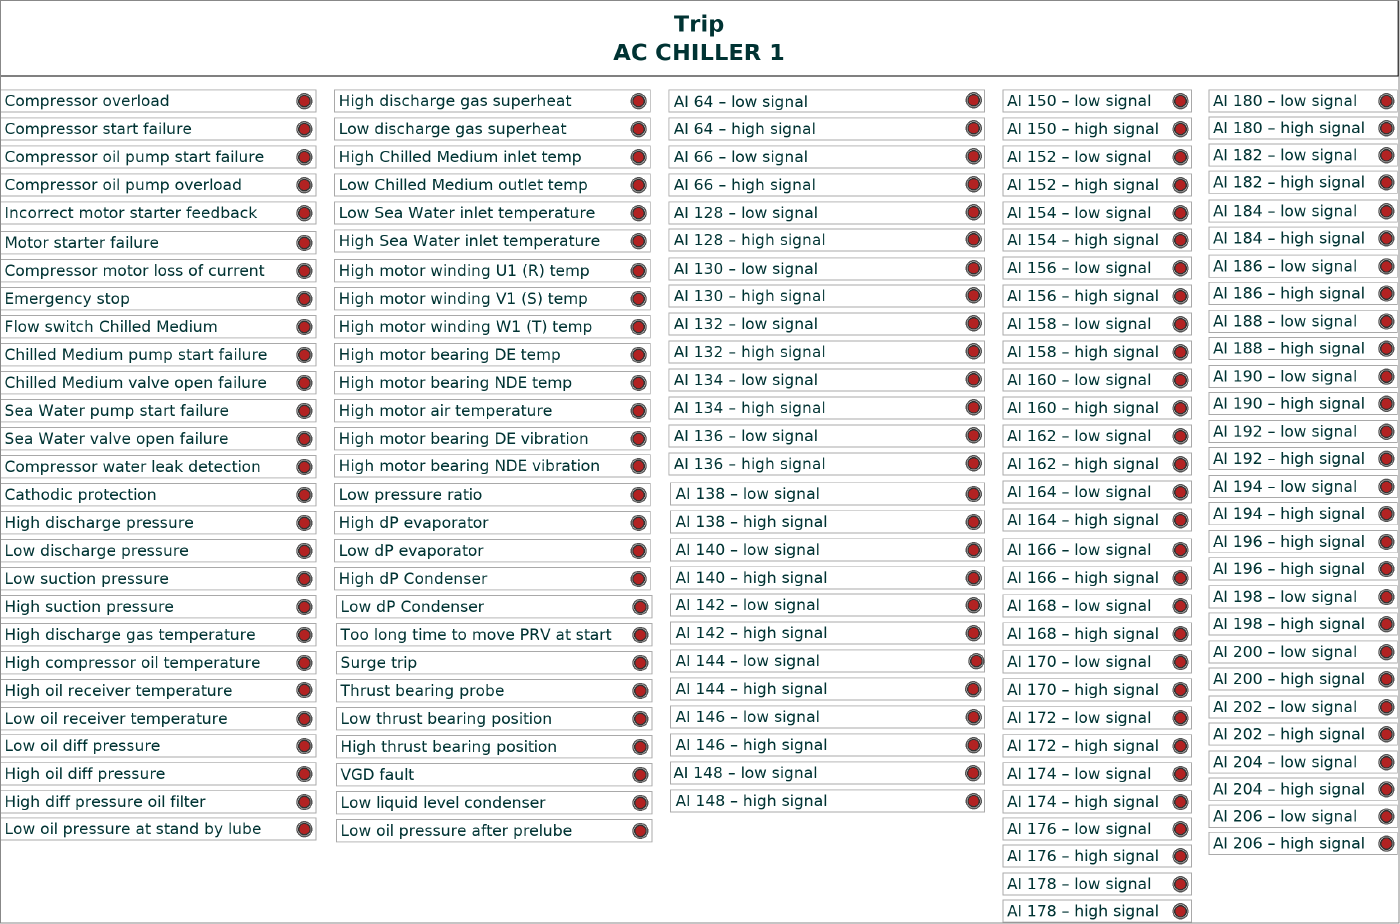
VISUALIZATION Chiller_1_Trip  // 1550x1023
    Rectangle (0,0 1548x84)
    Label (318,7 912x70), "Trip AC CHILLER 1"
    Rectangle (0,99 350x25)
    Label (2,101 319x21), "Compressor overload"
    Lamp1 (326,102 22x20), variable: Chiller_1.T_Overload_compressor_motor, style: Lamp-Lamp1-Red
    Rectangle (0,130 350x25)
    Label (2,132 319x21), "Compressor start failure"
    Lamp1 (326,133 22x20), variable: Chiller_1.T_Starter_failure_trip, style: Lamp-Lamp1-Red
    Rectangle (0,161 350x25)
    Label (2,163 319x21), "Compressor oil pump start failure"
    Lamp1 (326,164 22x20), variable: Chiller_1.T_Oil_pump_running_failure, style: Lamp-Lamp1-Red
    Rectangle (0,192 350x25)
    Label (2,194 319x21), "Compressor oil pump overload"
    Lamp1 (326,195 22x20), variable: Chiller_1.T_Overload_oil_pump_motor, style: Lamp-Lamp1-Red
    Rectangle (0,223 350x25)
    Label (2,225 319x21), "Incorrect motor starter feedback"
    Lamp1 (326,226 22x20), variable: Chiller_1.T_Compressor_running_failure, style: Lamp-Lamp1-Red
    Rectangle (370,535 350x25)
    Label (372,537 319x21), "Low pressure ratio"
    Lamp1 (696,538 22x20), variable: Chiller_1.T_Low_press_ratio, style: Lamp-Lamp1-Red
    Rectangle (370,566 350x25)
    Label (372,568 319x21), "High dP evaporator"
    Lamp1 (696,569 22x20), variable: Chiller_1.T_High_CW_dP, style: Lamp-Lamp1-Red
    Rectangle (370,597 350x25)
    Label (372,599 319x21), "Low dP evaporator"
    Lamp1 (696,600 22x20), variable: Chiller_1.T_Low_CW_dP, style: Lamp-Lamp1-Red
    Rectangle (370,628 350x25)
    Label (372,630 319x21), "High dP Condenser"
    Lamp1 (696,631 22x20), variable: Chiller_1.T_High_SW_dP, style: Lamp-Lamp1-Red
    Rectangle (0,256 350x25)
    Label (2,258 319x21), "Motor starter failure"
    Lamp1 (326,259 22x20), variable: Chiller_1.T_Motorstarter_failure, style: Lamp-Lamp1-Red
    Rectangle (0,287 350x25)
    Label (2,289 319x21), "Compressor motor loss of current"
    Lamp1 (326,290 22x20), variable: Chiller_1.T_Comp_motor_power_loss, style: Lamp-Lamp1-Red
    Rectangle (0,318 350x25)
    Label (2,320 319x21), "Emergency stop"
    Lamp1 (326,321 22x20), variable: Chiller_1.T_Emergency_stop, style: Lamp-Lamp1-Red
    Rectangle (0,349 350x25)
    Label (2,351 319x21), "Flow switch Chilled Medium"
    Lamp1 (326,352 22x20), variable: Chiller_1.T_Flow_switch_FT01, style: Lamp-Lamp1-Red
    Rectangle (0,380 350x25)
    Label (2,382 319x21), "Chilled Medium pump start failure"
    Lamp1 (326,383 22x20), variable: Chiller_1.T_Chilled_pump_run_failure, style: Lamp-Lamp1-Red
    Rectangle (0,411 350x25)
    Label (2,413 319x21), "Chilled Medium valve open failure"
    Lamp1 (326,414 22x20), variable: Chiller_1.T_CW_valveopen_failure, style: Lamp-Lamp1-Red
    Rectangle (0,442 350x25)
    Label (2,444 319x21), "Sea Water pump start failure"
    Lamp1 (326,445 22x20), variable: Chiller_1.T_Sea_water_pump_run_failure, style: Lamp-Lamp1-Red
    Rectangle (0,473 350x25)
    Label (2,475 319x21), "Sea Water valve open failure"
    Lamp1 (326,476 22x20), variable: Chiller_1.T_SW_valveopen_failure, style: Lamp-Lamp1-Red
    Rectangle (0,504 350x25)
    Label (2,506 319x21), "Compressor water leak detection"
    Lamp1 (326,507 22x20), variable: Chiller_1.T_Comp_motor_leak_detection, style: Lamp-Lamp1-Red
    Rectangle (0,535 350x25)
    Label (2,537 319x21), "Cathodic protection"
    Lamp1 (326,538 22x20), variable: Chiller_1.T_Cathodic_protect_sys_alarm, style: Lamp-Lamp1-Red
    Rectangle (0,566 350x25)
    Label (2,568 319x21), "High discharge pressure"
    Lamp1 (326,569 22x20), variable: Chiller_1.T_High_discharge_pressure, style: Lamp-Lamp1-Red
    Rectangle (0,597 350x25)
    Label (2,599 319x21), "Low discharge pressure"
    Lamp1 (326,600 22x20), variable: Chiller_1.T_Low_discharge_pressure, style: Lamp-Lamp1-Red
    Rectangle (0,659 350x25)
    Label (2,661 319x21), "High suction pressure"
    Lamp1 (326,662 22x20), variable: Chiller_1.T_High_suction_pressure, style: Lamp-Lamp1-Red
    Rectangle (0,628 350x25)
    Label (2,630 319x21), "Low suction pressure"
    Lamp1 (326,631 22x20), variable: Chiller_1.T_Low_suction_pressure, style: Lamp-Lamp1-Red
    Rectangle (0,690 350x25)
    Label (2,692 319x21), "High discharge gas temperature"
    Lamp1 (326,693 22x20), variable: Chiller_1.T_High_discharge_temp, style: Lamp-Lamp1-Red
    Rectangle (0,721 350x25)
    Label (2,723 319x21), "High compressor oil temperature"
    Lamp1 (326,724 22x20), variable: Chiller_1.T_High_temp_oil_inlet_comp, style: Lamp-Lamp1-Red
    Rectangle (0,752 350x25)
    Label (2,754 319x21), "High oil receiver temperature"
    Rectangle (0,813 350x25)
    Label (2,815 319x21), "Low oil diff pressure"
    Lamp1 (326,816 22x20), variable: Chiller_1.T_Low_oil_diff_pressure, style: Lamp-Lamp1-Red
    Rectangle (0,844 350x25)
    Label (2,846 319x21), "High oil diff pressure"
    Lamp1 (326,847 22x20), variable: Chiller_1.T_High_diff_oil_pressure, style: Lamp-Lamp1-Red
    Rectangle (0,875 350x25)
    Label (2,877 319x21), "High diff pressure oil filter"
    Lamp1 (326,878 22x20), variable: Chiller_1.T_High_oil_filter_diff_press, style: Lamp-Lamp1-Red
    Rectangle (0,783 350x25)
    Label (2,785 319x21), "Low oil receiver temperature"
    Lamp1 (326,786 22x20), variable: Chiller_1.T_Low_temp_oil_receiver, style: Lamp-Lamp1-Red
    Rectangle (370,99 350x25)
    Label (372,101 319x21), "High discharge gas superheat"
    Lamp1 (696,102 22x20), variable: Chiller_1.T_High_disch_superheat, style: Lamp-Lamp1-Red
    Rectangle (370,130 350x25)
    Label (372,132 319x21), "Low discharge gas superheat"
    Lamp1 (696,133 22x20), variable: Chiller_1.T_Low_disch_superheat, style: Lamp-Lamp1-Red
    Rectangle (370,161 350x25)
    Label (372,163 319x21), "High Chilled Medium inlet temp"
    Lamp1 (696,164 22x20), variable: Chiller_1.T_High_CW_inlet_temp, style: Lamp-Lamp1-Red
    Rectangle (370,192 350x25)
    Label (372,194 319x21), "Low Chilled Medium outlet temp"
    Lamp1 (696,195 22x20), variable: Chiller_1.T_Low_CW_outlet_temp, style: Lamp-Lamp1-Red
    Rectangle (370,223 350x25)
    Label (372,225 319x21), "Low Sea Water inlet temperature"
    Lamp1 (696,226 22x20), variable: Chiller_1.T_Low_SW_inlet_temp, style: Lamp-Lamp1-Red
    Rectangle (370,254 350x25)
    Label (372,256 319x21), "High Sea Water inlet temperature"
    Lamp1 (696,257 22x20), variable: Chiller_1.T_High_SW_inlet_temp, style: Lamp-Lamp1-Red
    Rectangle (370,503 350x25)
    Label (372,505 319x21), "High motor bearing NDE vibration"
    Lamp1 (696,506 22x20), variable: Chiller_1.T_High_comp_mot_NDE_bear_vib, style: Lamp-Lamp1-Red
    Rectangle (370,287 350x25)
    Label (372,289 319x21), "High motor winding U1 (R) temp"
    Lamp1 (696,290 22x20), variable: Chiller_1.T_High_motor_wind_temp_R, style: Lamp-Lamp1-Red
    Rectangle (370,318 350x25)
    Label (372,320 319x21), "High motor winding V1 (S) temp"
    Lamp1 (696,321 22x20), variable: Chiller_1.T_High_motor_wind_temp_S, style: Lamp-Lamp1-Red
    Rectangle (370,349 350x25)
    Label (372,351 319x21), "High motor winding W1 (T) temp"
    Lamp1 (696,352 22x20), variable: Chiller_1.T_High_motor_wind_temp_T, style: Lamp-Lamp1-Red
    Rectangle (370,380 350x25)
    Label (372,382 319x21), "High motor bearing DE temp"
    Lamp1 (696,383 22x20), variable: Chiller_1.T_High_comp_mot_DE_bear_temp, style: Lamp-Lamp1-Red
    Rectangle (370,411 350x25)
    Label (372,413 319x21), "High motor bearing NDE temp"
    Lamp1 (696,414 22x20), variable: Chiller_1.T_High_comp_mot_NDE_bear_temp, style: Lamp-Lamp1-Red
    Rectangle (370,442 350x25)
    Label (372,444 319x21), "High motor air temperature"
    Lamp1 (696,445 22x20), variable: Chiller_1.T_High_motor_air_temp, style: Lamp-Lamp1-Red
    Rectangle (370,473 350x25)
    Label (372,475 319x21), "High motor bearing DE vibration"
    Lamp1 (696,476 22x20), variable: Chiller_1.T_High_comp_mot_DE_bear_vib, style: Lamp-Lamp1-Red
    Rectangle (372,659 350x25)
    Label (374,661 319x21), "Low dP Condenser"
    Lamp1 (698,662 22x20), variable: Chiller_1.T_Low_SW_dP, style: Lamp-Lamp1-Red
    Rectangle (372,690 350x25)
    Label (374,692 319x21), "Too long time to move PRV at start"
    Lamp1 (698,693 22x20), variable: Chiller_1.T_Long_time_PRV, style: Lamp-Lamp1-Red
    Rectangle (372,721 350x25)
    Label (374,723 319x21), "Surge trip"
    Lamp1 (698,724 22x20), variable: Chiller_1.T_Surge_detection, style: Lamp-Lamp1-Red
    Rectangle (372,752 350x25)
    Label (374,754 319x21), "Thrust bearing probe"
    Lamp1 (698,755 22x20), variable: Chiller_1.T_Comp_thrust_bearing_position, style: Lamp-Lamp1-Red
    Rectangle (372,783 350x25)
    Label (374,785 319x21), "Low thrust bearing position"
    Lamp1 (698,786 22x20), variable: Chiller_1.T_Comp_thrust_neg_move, style: Lamp-Lamp1-Red
    Rectangle (372,814 350x25)
    Label (374,816 319x21), "High thrust bearing position"
    Lamp1 (698,817 22x20), variable: Chiller_1.T_Comp_thrust_pos_move, style: Lamp-Lamp1-Red
    Rectangle (372,845 350x25)
    Label (374,847 319x21), "VGD fault"
    Lamp1 (698,848 22x20), variable: Chiller_1.T_VGD_fault, style: Lamp-Lamp1-Red
    Rectangle (372,876 350x25)
    Label (374,878 319x21), "Low liquid level condenser"
    Lamp1 (698,879 22x20), variable: Chiller_1.T_Low_liquid_level, style: Lamp-Lamp1-Red
    Rectangle (372,907 350x25)
    Label (374,909 319x21), "Low oil pressure after prelube"
    Lamp1 (698,910 22x20), variable: Chiller_1.T_Low_oilpress_prelube, style: Lamp-Lamp1-Red
    Rectangle (1110,99 209x25)
    Rectangle (1110,130 209x25)
    Rectangle (1110,161 209x25)
    Rectangle (1110,192 209x25)
    Rectangle (1110,223 209x25)
    Lamp1 (1296,102 22x20), variable: Chiller_1.T_Sensor_low_signal_AI_150, style: Lamp-Lamp1-Red
    Lamp1 (1296,133 22x20), variable: Chiller_1.T_Sensor_high_signal_AI_150, style: Lamp-Lamp1-Red
    Lamp1 (1296,164 22x20), variable: Chiller_1.T_Sensor_low_signal_AI_152, style: Lamp-Lamp1-Red
    Lamp1 (1296,195 22x20), variable: Chiller_1.T_Sensor_high_signal_AI_152, style: Lamp-Lamp1-Red
    Label (1112,101 179x21), "AI 150 – low signal"
    Label (1112,132 179x21), "AI 150 – high signal"
    Label (1112,163 179x21), "AI 152 – low signal"
    Label (1112,194 179x21), "AI 152 – high signal"
    Label (1112,225 179x21), "AI 154 – low signal"
    Lamp1 (1296,226 22x20), variable: Chiller_1.T_Sensor_low_signal_AI_154, style: Lamp-Lamp1-Red
    Rectangle (1110,253 209x25)
    Label (1112,255 179x21), "AI 154 – high signal"
    Lamp1 (1296,256 22x20), variable: Chiller_1.T_Sensor_high_signal_AI_154, style: Lamp-Lamp1-Red
    Rectangle (1110,284 209x25)
    Rectangle (1110,315 209x25)
    Rectangle (1110,346 209x25)
    Rectangle (1110,377 209x25)
    Rectangle (1110,408 209x25)
    Rectangle (1110,439 209x25)
    Rectangle (1110,470 209x25)
    Rectangle (1110,501 209x25)
    Rectangle (1110,532 209x25)
    Rectangle (1110,563 209x25)
    Rectangle (1110,596 209x25)
    Rectangle (1110,627 209x25)
    Lamp1 (1296,287 22x20), variable: Chiller_1.T_Sensor_low_signal_AI_156, style: Lamp-Lamp1-Red
    Lamp1 (1296,318 22x20), variable: Chiller_1.T_Sensor_high_signal_AI_156, style: Lamp-Lamp1-Red
    Lamp1 (1296,349 22x20), variable: Chiller_1.T_Sensor_low_signal_AI_158, style: Lamp-Lamp1-Red
    Lamp1 (1296,380 22x20), variable: Chiller_1.T_Sensor_high_signal_AI_158, style: Lamp-Lamp1-Red
    Lamp1 (1296,411 22x20), variable: Chiller_1.T_Sensor_low_signal_AI_160, style: Lamp-Lamp1-Red
    Lamp1 (1296,442 22x20), variable: Chiller_1.T_Sensor_high_signal_AI_160, style: Lamp-Lamp1-Red
    Lamp1 (1296,473 22x20), variable: Chiller_1.T_Sensor_low_signal_AI_162, style: Lamp-Lamp1-Red
    Lamp1 (1296,504 22x20), variable: Chiller_1.T_Sensor_high_signal_AI_162, style: Lamp-Lamp1-Red
    Lamp1 (1296,535 22x20), variable: Chiller_1.T_Sensor_low_signal_AI_164, style: Lamp-Lamp1-Red
    Lamp1 (1296,566 22x20), variable: Chiller_1.T_Sensor_high_signal_AI_164, style: Lamp-Lamp1-Red
    Lamp1 (1296,599 22x20), variable: Chiller_1.T_Sensor_low_signal_AI_166, style: Lamp-Lamp1-Red
    Lamp1 (1296,630 22x20), variable: Chiller_1.T_Sensor_high_signal_AI_166, style: Lamp-Lamp1-Red
    Label (1112,286 179x21), "AI 156 – low signal"
    Label (1112,317 179x21), "AI 156 – high signal"
    Label (1112,348 179x21), "AI 158 – low signal"
    Label (1112,379 179x21), "AI 158 – high signal"
    Label (1112,410 179x21), "AI 160 – low signal"
    Label (1112,441 179x21), "AI 160 – high signal"
    Label (1112,472 179x21), "AI 162 – low signal"
    Label (1112,503 179x21), "AI 162 – high signal"
    Label (1112,534 179x21), "AI 164 – low signal"
    Label (1112,565 179x21), "AI 164 – high signal"
    Label (1112,598 179x21), "AI 166 – low signal"
    Label (1112,629 179x21), "AI 166 – high signal"
    Rectangle (1110,782 209x25)
    Rectangle (1110,658 209x25)
    Rectangle (1110,689 209x25)
    Rectangle (1110,720 209x25)
    Rectangle (1110,751 209x25)
    Rectangle (1110,813 209x25)
    Rectangle (1110,844 209x25)
    Rectangle (1110,875 209x25)
    Rectangle (1110,935 209x25)
    Rectangle (1110,996 209x25)
    Lamp1 (1296,785 22x20), variable: Chiller_1.T_Sensor_low_signal_AI_172, style: Lamp-Lamp1-Red
    Lamp1 (1296,661 22x20), variable: Chiller_1.T_Sensor_low_signal_AI_168, style: Lamp-Lamp1-Red
    Lamp1 (1296,692 22x20), variable: Chiller_1.T_Sensor_high_signal_AI_168, style: Lamp-Lamp1-Red
    Lamp1 (1296,723 22x20), variable: Chiller_1.T_Sensor_low_signal_AI_170, style: Lamp-Lamp1-Red
    Lamp1 (1296,754 22x20), variable: Chiller_1.T_Sensor_high_signal_AI_170, style: Lamp-Lamp1-Red
    Lamp1 (1296,816 22x20), variable: Chiller_1.T_Sensor_high_signal_AI_172, style: Lamp-Lamp1-Red
    Lamp1 (1296,847 22x20), variable: Chiller_1.T_Sensor_low_signal_AI_174, style: Lamp-Lamp1-Red
    Lamp1 (1296,878 22x20), variable: Chiller_1.T_Sensor_high_signal_AI_174, style: Lamp-Lamp1-Red
    Lamp1 (1296,938 22x20), variable: Chiller_1.T_Sensor_high_signal_AI_176, style: Lamp-Lamp1-Red
    Lamp1 (1296,999 22x20), variable: Chiller_1.T_Sensor_high_signal_AI_178, style: Lamp-Lamp1-Red
    Label (1112,784 179x21), "AI 172 – low signal"
    Label (1112,660 179x21), "AI 168 – low signal"
    Label (1112,691 179x21), "AI 168 – high signal"
    Label (1112,722 179x21), "AI 170 – low signal"
    Label (1112,753 179x21), "AI 170 – high signal"
    Label (1112,815 179x21), "AI 172 – high signal"
    Label (1112,846 179x21), "AI 174 – low signal"
    Label (1112,877 179x21), "AI 174 – high signal"
    Label (1112,937 179x21), "AI 176 – high signal"
    Label (1112,998 179x21), "AI 178 – high signal"
    Rectangle (740,192 350x25)
    Rectangle (740,99 350x25)
    Rectangle (740,130 350x25)
    Rectangle (740,161 350x25)
    Label (743,194 298x21), "AI 66 – high signal"
    Label (743,102 298x21), "AI 64 – low signal"
    Label (743,132 298x21), "AI 64 – high signal"
    Label (743,163 298x21), "AI 66 – low signal"
    Lamp1 (1066,194 24x20), variable: Chiller_1.T_Sensor_high_signal_AI_66, style: Lamp-Lamp1-Red
    Lamp1 (1066,101 24x20), variable: Chiller_1.T_Sensor_low_signal_AI_64, style: Lamp-Lamp1-Red
    Lamp1 (1066,132 24x20), variable: Chiller_1.T_Sensor_high_signal_AI_64, style: Lamp-Lamp1-Red
    Lamp1 (1066,163 24x20), variable: Chiller_1.T_Sensor_low_signal_AI_66, style: Lamp-Lamp1-Red
    Rectangle (740,346 350x25)
    Rectangle (740,377 350x25)
    Rectangle (740,408 350x25)
    Rectangle (740,439 350x25)
    Rectangle (740,470 350x25)
    Rectangle (740,501 350x25)
    Label (743,348 299x21), "AI 132 – low signal"
    Label (743,379 299x21), "AI 132 – high signal"
    Label (743,410 299x21), "AI 134 – low signal"
    Label (743,441 299x21), "AI 134 – high signal"
    Label (743,472 299x21), "AI 136 – low signal"
    Label (743,503 299x21), "AI 136 – high signal"
    Rectangle (740,315 350x25)
    Rectangle (740,223 350x25)
    Rectangle (740,253 350x25)
    Rectangle (740,285 350x25)
    Label (743,225 298x21), "AI 128 – low signal"
    Label (743,255 298x21), "AI 128 – high signal"
    Label (743,287 298x21), "AI 130 – low signal"
    Label (743,317 298x21), "AI 130 – high signal"
    Lamp1 (1066,348 24x20), variable: Chiller_1.T_Sensor_low_signal_AI_132, style: Lamp-Lamp1-Red
    Lamp1 (1066,379 24x20), variable: Chiller_1.T_Sensor_high_signal_AI_132, style: Lamp-Lamp1-Red
    Lamp1 (1066,410 24x20), variable: Chiller_1.T_Sensor_low_signal_AI_134, style: Lamp-Lamp1-Red
    Lamp1 (1066,441 24x20), variable: Chiller_1.T_Sensor_high_signal_AI_134, style: Lamp-Lamp1-Red
    Lamp1 (1066,472 24x20), variable: Chiller_1.T_Sensor_low_signal_AI_136, style: Lamp-Lamp1-Red
    Lamp1 (1066,503 24x20), variable: Chiller_1.T_Sensor_high_signal_AI_136, style: Lamp-Lamp1-Red
    Lamp1 (1066,225 24x20), variable: Chiller_1.T_Sensor_low_signal_AI_128, style: Lamp-Lamp1-Red
    Lamp1 (1066,255 24x20), variable: Chiller_1.T_Sensor_high_signal_AI_128, style: Lamp-Lamp1-Red
    Lamp1 (1066,287 24x20), variable: Chiller_1.T_Sensor_low_signal_AI_130, style: Lamp-Lamp1-Red
    Lamp1 (1066,317 24x20), variable: Chiller_1.T_Sensor_high_signal_AI_130, style: Lamp-Lamp1-Red
    Rectangle (742,843 348x25)
    Rectangle (742,627 348x25)
    Rectangle (742,657 348x25)
    Rectangle (742,688 348x25)
    Rectangle (742,719 348x25)
    Rectangle (742,750 348x25)
    Rectangle (742,781 348x25)
    Rectangle (742,812 348x25)
    Rectangle (742,874 348x25)
    Label (737,845 298x21), "AI 148 – low signal"
    Label (745,629 298x21), "AI 140 – high signal"
    Label (745,659 298x21), "AI 142 – low signal"
    Label (745,690 298x21), "AI 142 – high signal"
    Label (745,721 298x21), "AI 144 – low signal"
    Label (745,752 298x21), "AI 144 – high signal"
    Label (745,783 298x21), "AI 146 – low signal"
    Label (745,814 298x21), "AI 146 – high signal"
    Label (745,876 298x21), "AI 148 – high signal"
    Rectangle (742,596 348x25)
    Label (745,598 298x21), "AI 140 – low signal"
    Rectangle (742,565 348x25)
    Label (745,567 298x21), "AI 138 – high signal"
    Rectangle (742,534 348x25)
    Lamp1 (1066,846 23x20), variable: Chiller_1.T_Sensor_low_signal_AI_148, style: Lamp-Lamp1-Red
    Lamp1 (1066,630 24x20), variable: Chiller_1.T_Sensor_high_signal_AI_140, style: Lamp-Lamp1-Red
    Lamp1 (1066,660 24x20), variable: Chiller_1.T_Sensor_low_signal_AI_142, style: Lamp-Lamp1-Red
    Lamp1 (1066,691 24x20), variable: Chiller_1.T_Sensor_high_signal_AI_142, style: Lamp-Lamp1-Red
    Lamp1 (1066,722 30x20), variable: Chiller_1.T_Sensor_low_signal_AI_144, style: Lamp-Lamp1-Red
    Lamp1 (1066,753 23x20), variable: Chiller_1.T_Sensor_high_signal_AI_144, style: Lamp-Lamp1-Red
    Lamp1 (1066,784 24x20), variable: Chiller_1.T_Sensor_low_signal_AI_146, style: Lamp-Lamp1-Red
    Lamp1 (1066,815 24x20), variable: Chiller_1.T_Sensor_high_signal_AI_146, style: Lamp-Lamp1-Red
    Lamp1 (1066,877 24x20), variable: Chiller_1.T_Sensor_high_signal_AI_148, style: Lamp-Lamp1-Red
    Lamp1 (1066,599 24x20), variable: Chiller_1.T_Sensor_low_signal_AI_140, style: Lamp-Lamp1-Red
    Lamp1 (1066,568 24x20), variable: Chiller_1.T_Sensor_high_signal_AI_138, style: Lamp-Lamp1-Red
    Lamp1 (1066,537 24x20), variable: Chiller_1.T_Sensor_low_signal_AI_138, style: Lamp-Lamp1-Red
    Label (745,536 298x21), "AI 138 – low signal"
    Lamp1 (326,754 22x20), variable: Chiller_1.T_High_temp_oil_receiver, style: Lamp-Lamp1-Red
    Rectangle (0,905 350x25)
    Label (2,907 319x21), "Low oil pressure at stand by lube"
    Lamp1 (326,908 22x20), variable: Chiller_1.T_Low_oilpress_standby, style: Lamp-Lamp1-Red
    Rectangle (1110,905 209x25)
    Lamp1 (1296,908 22x20), variable: Chiller_1.T_Sensor_low_signal_AI_176, style: Lamp-Lamp1-Red
    Label (1112,907 179x21), "AI 176 – low signal"
    Rectangle (1110,966 209x25)
    Lamp1 (1296,969 22x20), variable: Chiller_1.T_Sensor_low_signal_AI_178, style: Lamp-Lamp1-Red
    Label (1112,968 179x21), "AI 178 – low signal"
    Rectangle (1338,129 209x25)
    Label (1340,131 179x21), "AI 180 – high signal"
    Lamp1 (1524,132 22x20), variable: Chiller_1.T_Sensor_high_signal_AI_180, style: Lamp-Lamp1-Red
    Rectangle (1338,189 209x25)
    Label (1340,191 179x21), "AI 182 – high signal"
    Lamp1 (1524,192 22x20), variable: Chiller_1.T_Sensor_high_signal_AI_182, style: Lamp-Lamp1-Red
    Rectangle (1338,495 209x25)
    Rectangle (1338,251 209x25)
    Rectangle (1338,312 209x25)
    Rectangle (1338,373 209x25)
    Rectangle (1338,434 209x25)
    Rectangle (1338,556 209x25)
    Rectangle (1338,617 209x25)
    Rectangle (1338,678 209x25)
    Rectangle (1338,739 209x25)
    Rectangle (1338,800 209x25)
    Rectangle (1338,861 209x25)
    Lamp1 (1524,498 22x20), variable: Chiller_1.T_Sensor_high_signal_AI_192, style: Lamp-Lamp1-Red
    Lamp1 (1524,254 22x20), variable: Chiller_1.T_Sensor_high_signal_AI_184, style: Lamp-Lamp1-Red
    Lamp1 (1524,315 22x20), variable: Chiller_1.T_Sensor_high_signal_AI_186, style: Lamp-Lamp1-Red
    Lamp1 (1524,376 22x20), variable: Chiller_1.T_Sensor_high_signal_AI_188, style: Lamp-Lamp1-Red
    Lamp1 (1524,437 22x20), variable: Chiller_1.T_Sensor_high_signal_AI_190, style: Lamp-Lamp1-Red
    Lamp1 (1524,559 22x20), variable: Chiller_1.T_Sensor_high_signal_AI_194, style: Lamp-Lamp1-Red
    Lamp1 (1524,620 22x20), variable: Chiller_1.T_Sensor_high_signal_AI_196, style: Lamp-Lamp1-Red
    Lamp1 (1524,681 22x20), variable: Chiller_1.T_Sensor_high_signal_AI_198, style: Lamp-Lamp1-Red
    Lamp1 (1524,742 22x20), variable: Chiller_1.T_Sensor_high_signal_AI_200, style: Lamp-Lamp1-Red
    Lamp1 (1524,803 22x20), variable: Chiller_1.T_Sensor_high_signal_AI_202, style: Lamp-Lamp1-Red
    Label (1340,497 179x21), "AI 192 – high signal"
    Label (1340,253 179x21), "AI 184 – high signal"
    Label (1340,314 179x21), "AI 186 – high signal"
    Label (1340,375 179x21), "AI 188 – high signal"
    Label (1340,436 179x21), "AI 190 – high signal"
    Label (1340,558 179x21), "AI 194 – high signal"
    Label (1340,619 179x21), "AI 196 – high signal"
    Label (1340,680 179x21), "AI 198 – high signal"
    Label (1340,741 179x21), "AI 200 – high signal"
    Label (1340,802 179x21), "AI 202 – high signal"
    Label (1340,863 179x21), "AI 204 – high signal"
    Lamp1 (1524,864 22x20), variable: Chiller_1.T_Sensor_high_signal_AI_204, style: Lamp-Lamp1-Red
    Rectangle (1338,921 209x25)
    Label (1340,923 179x21), "AI 206 – high signal"
    Lamp1 (1524,924 22x20), variable: Chiller_1.T_Sensor_high_signal_AI_206, style: Lamp-Lamp1-Red
    Rectangle (1338,99 209x25)
    Label (1340,101 179x21), "AI 180 – low signal"
    Lamp1 (1524,102 22x20), variable: Chiller_1.T_Sensor_low_signal_AI_180, style: Lamp-Lamp1-Red
    Rectangle (1338,159 209x25)
    Label (1340,161 179x21), "AI 182 – low signal"
    Lamp1 (1524,162 22x20), variable: Chiller_1.T_Sensor_low_signal_AI_182, style: Lamp-Lamp1-Red
    Rectangle (1338,221 209x25)
    Lamp1 (1524,224 22x20), variable: Chiller_1.T_Sensor_low_signal_AI_184, style: Lamp-Lamp1-Red
    Label (1340,223 179x21), "AI 184 – low signal"
    Rectangle (1338,282 209x25)
    Lamp1 (1524,285 22x20), variable: Chiller_1.T_Sensor_low_signal_AI_186, style: Lamp-Lamp1-Red
    Label (1340,284 179x21), "AI 186 – low signal"
    Rectangle (1338,343 209x25)
    Lamp1 (1524,346 22x20), variable: Chiller_1.T_Sensor_low_signal_AI_188, style: Lamp-Lamp1-Red
    Label (1340,345 179x21), "AI 188 – low signal"
    Rectangle (1338,404 209x25)
    Lamp1 (1524,407 22x20), variable: Chiller_1.T_Sensor_low_signal_AI_190, style: Lamp-Lamp1-Red
    Label (1340,406 179x21), "AI 190 – low signal"
    Rectangle (1338,465 209x25)
    Lamp1 (1524,468 22x20), variable: Chiller_1.T_Sensor_low_signal_AI_192, style: Lamp-Lamp1-Red
    Label (1340,467 179x21), "AI 192 – low signal"
    Rectangle (1338,526 209x25)
    Lamp1 (1524,529 22x20), variable: Chiller_1.T_Sensor_low_signal_AI_194, style: Lamp-Lamp1-Red
    Label (1340,528 179x21), "AI 194 – low signal"
    Rectangle (1338,587 209x25)
    Lamp1 (1524,590 22x20), variable: Chiller_1.T_Sensor_low_signal_AI_196, style: Lamp-Lamp1-Red
    Label (1340,589 179x21), "AI 196 – high signal"
    Rectangle (1338,648 209x25)
    Lamp1 (1524,651 22x20), variable: Chiller_1.T_Sensor_low_signal_AI_198, style: Lamp-Lamp1-Red
    Label (1340,650 179x21), "AI 198 – low signal"
    Rectangle (1338,709 209x25)
    Lamp1 (1524,712 22x20), variable: Chiller_1.T_Sensor_low_signal_AI_200, style: Lamp-Lamp1-Red
    Label (1340,711 179x21), "AI 200 – low signal"
    Rectangle (1338,770 209x25)
    Lamp1 (1524,773 22x20), variable: Chiller_1.T_Sensor_low_signal_AI_202, style: Lamp-Lamp1-Red
    Label (1340,772 179x21), "AI 202 – low signal"
    Rectangle (1338,831 209x25)
    Label (1340,833 179x21), "AI 204 – low signal"
    Lamp1 (1524,834 22x20), variable: Chiller_1.T_Sensor_low_signal_AI_204, style: Lamp-Lamp1-Red
    Rectangle (1338,891 209x25)
    Label (1340,893 179x21), "AI 206 – low signal"
    Lamp1 (1524,894 22x20), variable: Chiller_1.T_Sensor_low_signal_AI_206, style: Lamp-Lamp1-Red
END_VISUALIZATION

